LIN {X 0,Y 472.027,Z 1230.388,A -85,B 0,C 180,E1 22778.158,E2 22778.158} C_VEL
LIN {X 0,Y 471.943,Z 1235.002,A -85,B 0,C 180,E1 22775.714,E2 22775.714} C_VEL
LIN {X 0,Y 471.913,Z 1237.961,A -85,B 0,C 180,E1 22773.279,E2 22773.279} C_VEL
LIN {X 0,Y 471.908,Z 1239.363,A -85,B 0,C 180,E1 22770.728,E2 22770.728} C_VEL
LIN {X 0,Y 471.903,Z 1239.099,A -85,B 0,C 180,E1 22768.3,E2 22768.3} C_VEL
LIN {X 0,Y 471.92,Z 1237.256,A -85,B 0,C 180,E1 22765.869,E2 22765.869} C_VEL
LIN {X 0,Y 471.966,Z 1233.719,A -85,B 0,C 180,E1 22763.431,E2 22763.431} C_VEL
LIN {X 0,Y 472.092,Z 1228.265,A -85,B 0,C 180,E1 22760.86,E2 22760.86} C_VEL
LIN {X 0,Y 472.392,Z 1221.418,A -85,B 0,C 180,E1 22758.4,E2 22758.4} C_VEL
LIN {X 0,Y 472.916,Z 1212.648,A -85,B 0,C 180,E1 22755.928,E2 22755.928} C_VEL
LIN {X 0,Y 473.639,Z 1202.902,A -85,B 0,C 180,E1 22753.694,E2 22753.694} C_VEL
LIN {X 0,Y 474.601,Z 1191.85,A -85,B 0,C 180,E1 22751.578,E2 22751.578} C_VEL
LIN {X 0,Y 475.854,Z 1178.616,A -85,B 0,C 180,E1 22749.457,E2 22749.457} C_VEL
LIN {X 0,Y 477.335,Z 1163.705,A -85,B 0,C 180,E1 22747.46,E2 22747.46} C_VEL
LIN {X 0,Y 478.876,Z 1148.153,A -85,B 0,C 180,E1 22745.712,E2 22745.712} C_VEL
LIN {X 0,Y 480.486,Z 1131.656,A -85,B 0,C 180,E1 22744.153,E2 22744.153} C_VEL
LIN {X 0,Y 482.07,Z 1114.027,A -85,B 0,C 180,E1 22742.763,E2 22742.763} C_VEL
LIN {X 0,Y 483.619,Z 1095.064,A -85,B 0,C 180,E1 22741.539,E2 22741.539} C_VEL
LIN {X 0,Y 484.935,Z 1076.494,A -85,B 0,C 180,E1 22740.578,E2 22740.578} C_VEL
LIN {X 0,Y 486.066,Z 1056.533,A -85,B 0,C 180,E1 22739.778,E2 22739.778} C_VEL
LIN {X 0,Y 486.911,Z 1035.363,A -85,B 0,C 180,E1 22739.175,E2 22739.175} C_VEL
LIN {X 0,Y 487.494,Z 1006.649,A -85,B 0,C 180,E1 22738.67,E2 22738.67} C_VEL
LIN {X 0,Y 491.036,Z 793.925,A -85,B 0,C 180,E1 22735.273,E2 22735.273} C_VEL
LIN {X 0,Y 485.904,Z 771.478,A -85,B 0,C 180,E1 22734.421,E2 22734.421} C_VEL
LIN {X 0,Y 487.066,Z 742.84,A -85,B 0,C 180,E1 22731.537,E2 22731.537} C_VEL
LIN {X 0,Y 488.498,Z 716.424,A -85,B 0,C 180,E1 22728.693,E2 22728.693} C_VEL
LIN {X 0,Y 481.564,Z 696.985,A -85,B 0,C 180,E1 22725.751,E2 22725.751} C_VEL
LIN {X 0,Y 475.833,Z 682.945,A -85,B 0,C 180,E1 22723.536,E2 22723.536} C_VEL
LIN {X 0,Y 472.971,Z 675.939,A -85,B 0,C 180,E1 22722.424,E2 22722.424} C_VEL
LIN {X 0,Y 472.97,Z 675.954,A -85,B 0,C 180,E1 22721.46,E2 22721.46} C_VEL
LIN {X 0,Y 474.113,Z 679.098,A -85,B 0,C 180,E1 22720.975,E2 22720.975} C_VEL
LIN {X 0,Y 480.996,Z 694.968,A -85,B 0,C 180,E1 22718.497,E2 22718.497} C_VEL
LIN {X 0,Y 488.174,Z 713.188,A -85,B 0,C 180,E1 22715.858,E2 22715.858} C_VEL
LIN {X 0,Y 489.067,Z 715.897,A -85,B 0,C 180,E1 22715.494,E2 22715.494} C_VEL
LIN {X 0,Y 486.393,Z 754.227,A -85,B 0,C 180,E1 22711.891,E2 22711.891} C_VEL
LIN {X 0,Y 483.773,Z 794.316,A -85,B 0,C 180,E1 22708.182,E2 22708.182} C_VEL
LIN {X 0,Y 481.248,Z 836.985,A -85,B 0,C 180,E1 22704.291,E2 22704.291} C_VEL
LIN {X 0,Y 480.539,Z 852.687,A -85,B 0,C 180,E1 22702.912,E2 22702.912} C_VEL
LIN {X 0,Y 481.743,Z 862.638,A -85,B 0,C 180,E1 22702.654,E2 22702.654} C_VEL
LIN {X 0,Y 478.978,Z 1022.625,A -85,B 0,C 180,E1 22699.905,E2 22699.905} C_VEL
LIN {X 0,Y 478.54,Z 1040.298,A -85,B 0,C 180,E1 22699.368,E2 22699.368} C_VEL
LIN {X 0,Y 477.926,Z 1057.004,A -85,B 0,C 180,E1 22698.634,E2 22698.634} C_VEL
LIN {X 0,Y 477.154,Z 1073.057,A -85,B 0,C 180,E1 22697.689,E2 22697.689} C_VEL
LIN {X 0,Y 476.271,Z 1088.379,A -85,B 0,C 180,E1 22696.527,E2 22696.527} C_VEL
LIN {X 0,Y 475.395,Z 1102.609,A -85,B 0,C 180,E1 22695.18,E2 22695.18} C_VEL
LIN {X 0,Y 474.55,Z 1115.691,A -85,B 0,C 180,E1 22693.65,E2 22693.65} C_VEL
LIN {X 0,Y 473.843,Z 1126.703,A -85,B 0,C 180,E1 22692.058,E2 22692.058} C_VEL
LIN {X 0,Y 473.206,Z 1137.011,A -85,B 0,C 180,E1 22690.224,E2 22690.224} C_VEL
LIN {X 0,Y 472.752,Z 1145.711,A -85,B 0,C 180,E1 22688.269,E2 22688.269} C_VEL
LIN {X 0,Y 472.48,Z 1152.378,A -85,B 0,C 180,E1 22686.318,E2 22686.318} C_VEL
LIN {X 0,Y 472.291,Z 1157.831,A -85,B 0,C 180,E1 22684.128,E2 22684.128} C_VEL
LIN {X 0,Y 472.226,Z 1161.226,A -85,B 0,C 180,E1 22682.011,E2 22682.011} C_VEL
LIN {X 0,Y 472.201,Z 1162.941,A -85,B 0,C 180,E1 22679.879,E2 22679.879} C_VEL
LIN {X 0,Y 472.231,Z 1162.833,A -85,B 0,C 180,E1 22677.573,E2 22677.573} C_VEL
LIN {X 0,Y 472.284,Z 1161.078,A -85,B 0,C 180,E1 22675.508,E2 22675.508} C_VEL
LIN {X 0,Y 472.422,Z 1157.73,A -85,B 0,C 180,E1 22673.438,E2 22673.438} C_VEL
LIN {X 0,Y 472.653,Z 1152.534,A -85,B 0,C 180,E1 22671.362,E2 22671.362} C_VEL
LIN {X 0,Y 473.024,Z 1145.419,A -85,B 0,C 180,E1 22669.28,E2 22669.28} C_VEL
LIN {X 0,Y 473.566,Z 1137.253,A -85,B 0,C 180,E1 22667.44,E2 22667.44} C_VEL
LIN {X 0,Y 474.243,Z 1127.651,A -85,B 0,C 180,E1 22665.72,E2 22665.72} C_VEL
LIN {X 0,Y 474.992,Z 1116.619,A -85,B 0,C 180,E1 22664.119,E2 22664.119} C_VEL
LIN {X 0,Y 475.86,Z 1104.113,A -85,B 0,C 180,E1 22662.641,E2 22662.641} C_VEL
LIN {X 0,Y 476.736,Z 1090.596,A -85,B 0,C 180,E1 22661.347,E2 22661.347} C_VEL
LIN {X 0,Y 477.533,Z 1075.977,A -85,B 0,C 180,E1 22660.236,E2 22660.236} C_VEL
LIN {X 0,Y 478.208,Z 1060.301,A -85,B 0,C 180,E1 22659.308,E2 22659.308} C_VEL
LIN {X 0,Y 478.738,Z 1043.983,A -85,B 0,C 180,E1 22658.586,E2 22658.586} C_VEL
LIN {X 0,Y 479.03,Z 1027.199,A -85,B 0,C 180,E1 22658.081,E2 22658.081} C_VEL
LIN {X 0,Y 481.097,Z 935.545,A -85,B 0,C 180,E1 22656.323,E2 22656.323} C_VEL
LIN {X 0,Y 483.696,Z 869.516,A -85,B 0,C 180,E1 22654.928,E2 22654.928} C_VEL
LIN {X 0,Y 486.372,Z 861.818,A -85,B 0,C 180,E1 22654.359,E2 22654.359} C_VEL
LIN {X 0,Y 491.455,Z 830.458,A -85,B 0,C 180,E1 22650.973,E2 22650.973} C_VEL
LIN {X 0,Y 496.727,Z 807.951,A -85,B 0,C 180,E1 22648.371,E2 22648.371} C_VEL
LIN {X 0,Y 502.512,Z 790.111,A -85,B 0,C 180,E1 22646.143,E2 22646.143} C_VEL
LIN {X 0,Y 508.797,Z 776.41,A -85,B 0,C 180,E1 22644.293,E2 22644.293} C_VEL
LIN {X 0,Y 509.848,Z 774.506,A -85,B 0,C 180,E1 22643.994,E2 22643.994} C_VEL
LIN {X 0,Y 502.789,Z 785.083,A -85,B 0,C 180,E1 22642.698,E2 22642.698} C_VEL
LIN {X 0,Y 498.164,Z 795.448,A -85,B 0,C 180,E1 22641.413,E2 22641.413} C_VEL
LIN {X 0,Y 495.854,Z 805.348,A -85,B 0,C 180,E1 22640.199,E2 22640.199} C_VEL
LIN {X 0,Y 495.553,Z 815.668,A -85,B 0,C 180,E1 22638.956,E2 22638.956} C_VEL
LIN {X 0,Y 497.374,Z 826.582,A -85,B 0,C 180,E1 22637.667,E2 22637.667} C_VEL
LIN {X 0,Y 501.457,Z 837.677,A -85,B 0,C 180,E1 22636.379,E2 22636.379} C_VEL
LIN {X 0,Y 507.651,Z 848.231,A -85,B 0,C 180,E1 22635.158,E2 22635.158} C_VEL
LIN {X 0,Y 515.78,Z 858.073,A -85,B 0,C 180,E1 22634.012,E2 22634.012} C_VEL
LIN {X 0,Y 525.907,Z 867.121,A -85,B 0,C 180,E1 22632.949,E2 22632.949} C_VEL
LIN {X 0,Y 537.102,Z 874.718,A -85,B 0,C 180,E1 22632.032,E2 22632.032} C_VEL
LIN {X 0,Y 549.32,Z 880.935,A -85,B 0,C 180,E1 22631.217,E2 22631.217} C_VEL
LIN {X 0,Y 556.729,Z 883.664,A -85,B 0,C 180,E1 22630.722,E2 22630.722} C_VEL
LIN {X 0,Y 559.457,Z 884.419,A -85,B 0,C 180,E1 22630.458,E2 22630.458} C_VEL
LIN {X 0,Y 556.641,Z 890.597,A -85,B 0,C 180,E1 22630.289,E2 22630.289} C_VEL
LIN {X 0,Y 545.031,Z 908.312,A -85,B 0,C 180,E1 22629.947,E2 22629.947} C_VEL
LIN {X 0,Y 525.372,Z 938.085,A -85,B 0,C 180,E1 22629.116,E2 22629.116} C_VEL
LIN {X 0,Y 515.376,Z 955.996,A -85,B 0,C 180,E1 22628.518,E2 22628.518} C_VEL
LIN {X 0,Y 509.372,Z 970.036,A -85,B 0,C 180,E1 22627.98,E2 22627.98} C_VEL
LIN {X 0,Y 506.831,Z 975.536,A -85,B 0,C 180,E1 22627.774,E2 22627.774} C_VEL
LIN {X 0,Y 500.091,Z 990.21,A -85,B 0,C 180,E1 22627.215,E2 22627.215} C_VEL
LIN {X 0,Y 492.099,Z 1013.905,A -85,B 0,C 180,E1 22626.175,E2 22626.175} C_VEL
LIN {X 0,Y 490.679,Z 1019.518,A -85,B 0,C 180,E1 22625.946,E2 22625.946} C_VEL
LIN {X 0,Y 490.022,Z 1029.861,A -85,B 0,C 180,E1 22625.815,E2 22625.815} C_VEL
LIN {X 0,Y 489.453,Z 1064.268,A -85,B 0,C 180,E1 22625.251,E2 22625.251} C_VEL
LIN {X 0,Y 488.525,Z 1088.169,A -85,B 0,C 180,E1 22624.651,E2 22624.651} C_VEL
LIN {X 0,Y 487.384,Z 1111.453,A -85,B 0,C 180,E1 22623.84,E2 22623.84} C_VEL
LIN {X 0,Y 486.067,Z 1134.154,A -85,B 0,C 180,E1 22622.822,E2 22622.822} C_VEL
LIN {X 0,Y 484.559,Z 1155.984,A -85,B 0,C 180,E1 22621.609,E2 22621.609} C_VEL
LIN {X 0,Y 482.968,Z 1176.918,A -85,B 0,C 180,E1 22620.204,E2 22620.204} C_VEL
LIN {X 0,Y 481.619,Z 1192.738,A -85,B 0,C 180,E1 22618.929,E2 22618.929} C_VEL
LIN {X 0,Y 480.163,Z 1206.829,A -85,B 0,C 180,E1 22617.535,E2 22617.535} C_VEL
LIN {X 0,Y 478.573,Z 1221.087,A -85,B 0,C 180,E1 22615.891,E2 22615.891} C_VEL
LIN {X 0,Y 477.202,Z 1233.662,A -85,B 0,C 180,E1 22614.247,E2 22614.247} C_VEL
LIN {X 0,Y 475.743,Z 1248.075,A -85,B 0,C 180,E1 22612.099,E2 22612.099} C_VEL
LIN {X 0,Y 474.509,Z 1260.921,A -85,B 0,C 180,E1 22609.832,E2 22609.832} C_VEL
LIN {X 0,Y 473.67,Z 1270.78,A -85,B 0,C 180,E1 22607.823,E2 22607.823} C_VEL
LIN {X 0,Y 472.974,Z 1280.325,A -85,B 0,C 180,E1 22605.574,E2 22605.574} C_VEL
LIN {X 0,Y 472.429,Z 1289.877,A -85,B 0,C 180,E1 22602.84,E2 22602.84} C_VEL
LIN {X 0,Y 472.149,Z 1296.436,A -85,B 0,C 180,E1 22600.494,E2 22600.494} C_VEL
LIN {X 0,Y 471.998,Z 1301.632,A -85,B 0,C 180,E1 22598.16,E2 22598.16} C_VEL
LIN {X 0,Y 471.927,Z 1306.121,A -85,B 0,C 180,E1 22595.349,E2 22595.349} C_VEL
LIN {X 0,Y 471.903,Z 1308.434,A -85,B 0,C 180,E1 22592.915,E2 22592.915} C_VEL
LIN {X 0,Y 471.896,Z 1309.388,A -85,B 0,C 180,E1 22590.608,E2 22590.608} C_VEL
LIN {X 0,Y 471.908,Z 1308.917,A -85,B 0,C 180,E1 22587.815,E2 22587.815} C_VEL
LIN {X 0,Y 471.918,Z 1306.943,A -85,B 0,C 180,E1 22585.383,E2 22585.383} C_VEL
LIN {X 0,Y 471.961,Z 1303.794,A -85,B 0,C 180,E1 22583.065,E2 22583.065} C_VEL
LIN {X 0,Y 472.071,Z 1299.112,A -85,B 0,C 180,E1 22580.614,E2 22580.614} C_VEL
LIN {X 0,Y 472.324,Z 1292.113,A -85,B 0,C 180,E1 22577.903,E2 22577.903} C_VEL
LIN {X 0,Y 472.718,Z 1284.471,A -85,B 0,C 180,E1 22575.548,E2 22575.548} C_VEL
LIN {X 0,Y 473.375,Z 1274.765,A -85,B 0,C 180,E1 22573.054,E2 22573.054} C_VEL
LIN {X 0,Y 474.273,Z 1263.528,A -85,B 0,C 180,E1 22570.672,E2 22570.672} C_VEL
LIN {X 0,Y 475.286,Z 1252.524,A -85,B 0,C 180,E1 22568.658,E2 22568.658} C_VEL
LIN {X 0,Y 476.669,Z 1239.071,A -85,B 0,C 180,E1 22566.514,E2 22566.514} C_VEL
LIN {X 0,Y 478.346,Z 1223.146,A -85,B 0,C 180,E1 22564.363,E2 22564.363} C_VEL
LIN {X 0,Y 479.836,Z 1209.702,A -85,B 0,C 180,E1 22562.782,E2 22562.782} C_VEL
LIN {X 0,Y 481.31,Z 1196.28,A -85,B 0,C 180,E1 22561.392,E2 22561.392} C_VEL
LIN {X 0,Y 483.032,Z 1177.605,A -85,B 0,C 180,E1 22559.802,E2 22559.802} C_VEL
LIN {X 0,Y 484.805,Z 1157.277,A -85,B 0,C 180,E1 22558.341,E2 22558.341} C_VEL
LIN {X 0,Y 486.575,Z 1135.76,A -85,B 0,C 180,E1 22557.055,E2 22557.055} C_VEL
LIN {X 0,Y 488.148,Z 1114.091,A -85,B 0,C 180,E1 22556.002,E2 22556.002} C_VEL
LIN {X 0,Y 489.575,Z 1091.135,A -85,B 0,C 180,E1 22555.128,E2 22555.128} C_VEL
LIN {X 0,Y 490.74,Z 1068.207,A -85,B 0,C 180,E1 22554.494,E2 22554.494} C_VEL
LIN {X 0,Y 491.441,Z 1041.848,A -85,B 0,C 180,E1 22554.015,E2 22554.015} C_VEL
LIN {X 0,Y 492.099,Z 1021.688,A -85,B 0,C 180,E1 22553.682,E2 22553.682} C_VEL
LIN {X 0,Y 497.028,Z 1006.052,A -85,B 0,C 180,E1 22552.952,E2 22552.952} C_VEL
LIN {X 0,Y 503.429,Z 988.405,A -85,B 0,C 180,E1 22552.208,E2 22552.208} C_VEL
LIN {X 0,Y 510.583,Z 973.055,A -85,B 0,C 180,E1 22551.7,E2 22551.7} C_VEL
LIN {X 0,Y 516.137,Z 959.333,A -85,B 0,C 180,E1 22551.195,E2 22551.195} C_VEL
LIN {X 0,Y 524.952,Z 942.125,A -85,B 0,C 180,E1 22550.707,E2 22550.707} C_VEL
LIN {X 0,Y 541.254,Z 914.948,A -85,B 0,C 180,E1 22550.133,E2 22550.133} C_VEL
LIN {X 0,Y 557.706,Z 888.615,A -85,B 0,C 180,E1 22549.67,E2 22549.67} C_VEL
LIN {X 0,Y 559.402,Z 884.287,A -85,B 0,C 180,E1 22549.528,E2 22549.528} C_VEL
LIN {X 0,Y 547.093,Z 880.541,A -85,B 0,C 180,E1 22548.372,E2 22548.372} C_VEL
LIN {X 0,Y 536.038,Z 875.106,A -85,B 0,C 180,E1 22547.143,E2 22547.143} C_VEL
LIN {X 0,Y 526.595,Z 868.26,A -85,B 0,C 180,E1 22545.866,E2 22545.866} C_VEL
LIN {X 0,Y 518.671,Z 860.097,A -85,B 0,C 180,E1 22544.563,E2 22544.563} C_VEL
LIN {X 0,Y 512.248,Z 850.667,A -85,B 0,C 180,E1 22543.245,E2 22543.245} C_VEL
LIN {X 0,Y 507.136,Z 839.468,A -85,B 0,C 180,E1 22541.865,E2 22541.865} C_VEL
LIN {X 0,Y 503.479,Z 826.201,A -85,B 0,C 180,E1 22540.42,E2 22540.42} C_VEL
LIN {X 0,Y 501.504,Z 811.016,A -85,B 0,C 180,E1 22538.964,E2 22538.964} C_VEL
LIN {X 0,Y 501.31,Z 794.305,A -85,B 0,C 180,E1 22537.54,E2 22537.54} C_VEL
LIN {X 0,Y 505.763,Z 740.56,A -85,B 0,C 180,E1 22533.413,E2 22533.413} C_VEL
LIN {X 0,Y 506.021,Z 736.154,A -85,B 0,C 180,E1 22533.049,E2 22533.049} C_VEL
LIN {X 0,Y 496.27,Z 718.046,A -85,B 0,C 180,E1 22529.977,E2 22529.977} C_VEL
LIN {X 0,Y 488.915,Z 704.66,A -85,B 0,C 180,E1 22527.528,E2 22527.528} C_VEL
LIN {X 0,Y 483.047,Z 694.382,A -85,B 0,C 180,E1 22525.501,E2 22525.501} C_VEL
LIN {X 0,Y 480.533,Z 689.941,A -85,B 0,C 180,E1 22524.591,E2 22524.591} C_VEL
LIN {X 0,Y 478.059,Z 685.483,A -85,B 0,C 180,E1 22523.676,E2 22523.676} C_VEL
LIN {X 0,Y 475.958,Z 681.627,A -85,B 0,C 180,E1 22522.869,E2 22522.869} C_VEL
LIN {X 0,Y 473.409,Z 677.657,A -85,B 0,C 180,E1 22521.952,E2 22521.952} C_VEL
LIN {X 0,Y 472.947,Z 675.821,A -85,B 0,C 180,E1 22521.648,E2 22521.648} C_VEL
LIN {X 0,Y 472.954,Z 675.824,A -85,B 0,C 180,E1 22517.978,E2 22517.978} C_VEL
LIN {X 0,Y 472.946,Z 675.824,A -85,B 0,C 180,E1 22514.321,E2 22514.321} C_VEL
LIN {X 0,Y 472.947,Z 675.824,A -85,B 0,C 180,E1 22510.722,E2 22510.722} C_VEL
LIN {X 0,Y 472.958,Z 675.82,A -85,B 0,C 180,E1 22507.043,E2 22507.043} C_VEL
LIN {X 0,Y 472.941,Z 675.824,A -85,B 0,C 180,E1 22503.393,E2 22503.393} C_VEL
LIN {X 0,Y 472.954,Z 675.821,A -85,B 0,C 180,E1 22499.757,E2 22499.757} C_VEL
LIN {X 0,Y 472.947,Z 675.821,A -85,B 0,C 180,E1 22496.121,E2 22496.121} C_VEL
LIN {X 0,Y 472.937,Z 675.825,A -85,B 0,C 180,E1 22492.468,E2 22492.468} C_VEL
LIN {X 0,Y 472.95,Z 675.822,A -85,B 0,C 180,E1 22488.908,E2 22488.908} C_VEL
LIN {X 0,Y 472.949,Z 675.823,A -85,B 0,C 180,E1 22485.304,E2 22485.304} C_VEL
LIN {X 0,Y 472.939,Z 675.821,A -85,B 0,C 180,E1 22481.639,E2 22481.639} C_VEL
LIN {X 0,Y 472.957,Z 675.821,A -85,B 0,C 180,E1 22478.026,E2 22478.026} C_VEL
LIN {X 0,Y 472.942,Z 675.823,A -85,B 0,C 180,E1 22474.316,E2 22474.316} C_VEL
LIN {X 0,Y 472.936,Z 675.784,A -85,B 0,C 180,E1 22470.766,E2 22470.766} C_VEL
LIN {X 0,Y 472.954,Z 675.822,A -85,B 0,C 180,E1 22467.234,E2 22467.234} C_VEL
LIN {X 0,Y 472.938,Z 675.8,A -85,B 0,C 180,E1 22463.553,E2 22463.553} C_VEL
LIN {X 0,Y 472.938,Z 675.802,A -85,B 0,C 180,E1 22460.006,E2 22460.006} C_VEL
LIN {X 0,Y 472.951,Z 675.825,A -85,B 0,C 180,E1 22456.433,E2 22456.433} C_VEL
LIN {X 0,Y 472.966,Z 675.939,A -85,B 0,C 180,E1 22454.184,E2 22454.184} C_VEL
LIN {X 0,Y 474.014,Z 678.945,A -85,B 0,C 180,E1 22453.83,E2 22453.83} C_VEL
LIN {X 0,Y 475.481,Z 681.845,A -85,B 0,C 180,E1 22453.442,E2 22453.442} C_VEL
LIN {X 0,Y 483.15,Z 698.3,A -85,B 0,C 180,E1 22451.304,E2 22451.304} C_VEL
LIN {X 0,Y 490.743,Z 716.812,A -85,B 0,C 180,E1 22449.08,E2 22449.08} C_VEL
LIN {X 0,Y 488.698,Z 760.843,A -85,B 0,C 180,E1 22445.884,E2 22445.884} C_VEL
LIN {X 0,Y 488.556,Z 770.502,A -85,B 0,C 180,E1 22445.256,E2 22445.256} C_VEL
LIN {X 0,Y 489.009,Z 773.268,A -85,B 0,C 180,E1 22445.169,E2 22445.169} C_VEL
LIN {X 0,Y 489.235,Z 779.807,A -85,B 0,C 180,E1 22445.034,E2 22445.034} C_VEL
LIN {X 0,Y 487.638,Z 789.743,A -85,B 0,C 180,E1 22444.991,E2 22444.991} C_VEL
LIN {X 0,Y 484.595,Z 804.217,A -85,B 0,C 180,E1 22444.989,E2 22444.989} C_VEL
LIN {X 0,Y 484.245,Z 808.717,A -85,B 0,C 180,E1 22444.938,E2 22444.938} C_VEL
LIN {X 0,Y 480.185,Z 1031.487,A -85,B 0,C 180,E1 22441.312,E2 22441.312} C_VEL
LIN {X 0,Y 479.366,Z 1052.367,A -85,B 0,C 180,E1 22440.762,E2 22440.762} C_VEL
LIN {X 0,Y 478.234,Z 1073.043,A -85,B 0,C 180,E1 22439.978,E2 22439.978} C_VEL
LIN {X 0,Y 476.872,Z 1092.041,A -85,B 0,C 180,E1 22439.034,E2 22439.034} C_VEL
LIN {X 0,Y 475.373,Z 1110.231,A -85,B 0,C 180,E1 22437.903,E2 22437.903} C_VEL
LIN {X 0,Y 473.655,Z 1128.403,A -85,B 0,C 180,E1 22436.516,E2 22436.516} C_VEL
LIN {X 0,Y 471.885,Z 1145.616,A -85,B 0,C 180,E1 22434.923,E2 22434.923} C_VEL
LIN {X 0,Y 470.228,Z 1160.946,A -85,B 0,C 180,E1 22433.23,E2 22433.23} C_VEL
LIN {X 0,Y 468.703,Z 1175.051,A -85,B 0,C 180,E1 22431.394,E2 22431.394} C_VEL
LIN {X 0,Y 467.317,Z 1188.383,A -85,B 0,C 180,E1 22429.342,E2 22429.342} C_VEL
LIN {X 0,Y 466.197,Z 1200.038,A -85,B 0,C 180,E1 22427.215,E2 22427.215} C_VEL
LIN {X 0,Y 465.312,Z 1210.434,A -85,B 0,C 180,E1 22424.942,E2 22424.942} C_VEL
LIN {X 0,Y 464.634,Z 1219.787,A -85,B 0,C 180,E1 22422.426,E2 22422.426} C_VEL
LIN {X 0,Y 464.237,Z 1227.132,A -85,B 0,C 180,E1 22419.921,E2 22419.921} C_VEL
LIN {X 0,Y 464.022,Z 1232.679,A -85,B 0,C 180,E1 22417.428,E2 22417.428} C_VEL
LIN {X 0,Y 463.939,Z 1236.571,A -85,B 0,C 180,E1 22414.945,E2 22414.945} C_VEL
LIN {X 0,Y 463.918,Z 1238.909,A -85,B 0,C 180,E1 22412.47,E2 22412.47} C_VEL
LIN {X 0,Y 463.917,Z 1239.729,A -85,B 0,C 180,E1 22409.999,E2 22409.999} C_VEL
LIN {X 0,Y 463.915,Z 1238.892,A -85,B 0,C 180,E1 22407.405,E2 22407.405} C_VEL
LIN {X 0,Y 463.94,Z 1236.53,A -85,B 0,C 180,E1 22404.93,E2 22404.93} C_VEL
LIN {X 0,Y 464.039,Z 1232.365,A -85,B 0,C 180,E1 22402.322,E2 22402.322} C_VEL
LIN {X 0,Y 464.255,Z 1226.654,A -85,B 0,C 180,E1 22399.814,E2 22399.814} C_VEL
LIN {X 0,Y 464.645,Z 1219.655,A -85,B 0,C 180,E1 22397.447,E2 22397.447} C_VEL
LIN {X 0,Y 465.28,Z 1210.794,A -85,B 0,C 180,E1 22395.056,E2 22395.056} C_VEL
LIN {X 0,Y 466.216,Z 1199.849,A -85,B 0,C 180,E1 22392.656,E2 22392.656} C_VEL
LIN {X 0,Y 467.356,Z 1188.005,A -85,B 0,C 180,E1 22390.503,E2 22390.503} C_VEL
LIN {X 0,Y 468.736,Z 1174.764,A -85,B 0,C 180,E1 22388.475,E2 22388.475} C_VEL
LIN {X 0,Y 470.373,Z 1159.524,A -85,B 0,C 180,E1 22386.511,E2 22386.511} C_VEL
LIN {X 0,Y 472.158,Z 1142.897,A -85,B 0,C 180,E1 22384.72,E2 22384.72} C_VEL
LIN {X 0,Y 473.89,Z 1125.851,A -85,B 0,C 180,E1 22383.188,E2 22383.188} C_VEL
LIN {X 0,Y 475.513,Z 1108.664,A -85,B 0,C 180,E1 22381.9,E2 22381.9} C_VEL
LIN {X 0,Y 477.041,Z 1090.144,A -85,B 0,C 180,E1 22380.767,E2 22380.767} C_VEL
LIN {X 0,Y 478.393,Z 1070.604,A -85,B 0,C 180,E1 22379.824,E2 22379.824} C_VEL
LIN {X 0,Y 479.447,Z 1050.707,A -85,B 0,C 180,E1 22379.095,E2 22379.095} C_VEL
LIN {X 0,Y 480.227,Z 1029.772,A -85,B 0,C 180,E1 22378.563,E2 22378.563} C_VEL
LIN {X 0,Y 484.468,Z 796.881,A -85,B 0,C 180,E1 22374.778,E2 22374.778} C_VEL
LIN {X 0,Y 483.819,Z 792.472,A -85,B 0,C 180,E1 22374.644,E2 22374.644} C_VEL
LIN {X 0,Y 479.103,Z 772.305,A -85,B 0,C 180,E1 22373.867,E2 22373.867} C_VEL
LIN {X 0,Y 480.243,Z 745.321,A -85,B 0,C 180,E1 22371.139,E2 22371.139} C_VEL
LIN {X 0,Y 481.659,Z 719.994,A -85,B 0,C 180,E1 22368.408,E2 22368.408} C_VEL
LIN {X 0,Y 474.936,Z 701.008,A -85,B 0,C 180,E1 22365.488,E2 22365.488} C_VEL
LIN {X 0,Y 469.094,Z 686.695,A -85,B 0,C 180,E1 22363.173,E2 22363.173} C_VEL
LIN {X 0,Y 466.014,Z 679.803,A -85,B 0,C 180,E1 22362.022,E2 22362.022} C_VEL
LIN {X 0,Y 465.799,Z 679.402,A -85,B 0,C 180,E1 22361.922,E2 22361.922} C_VEL
LIN {X 0,Y 468.625,Z 685.422,A -85,B 0,C 180,E1 22360.921,E2 22360.921} C_VEL
LIN {X 0,Y 476.2,Z 703.373,A -85,B 0,C 180,E1 22358.12,E2 22358.12} C_VEL
LIN {X 0,Y 482.247,Z 719.132,A -85,B 0,C 180,E1 22355.838,E2 22355.838} C_VEL
LIN {X 0,Y 479.481,Z 756.766,A -85,B 0,C 180,E1 22352.265,E2 22352.265} C_VEL
LIN {X 0,Y 476.721,Z 797.118,A -85,B 0,C 180,E1 22348.502,E2 22348.502} C_VEL
LIN {X 0,Y 474.03,Z 840.018,A -85,B 0,C 180,E1 22344.553,E2 22344.553} C_VEL
LIN {X 0,Y 473.384,Z 853.662,A -85,B 0,C 180,E1 22343.346,E2 22343.346} C_VEL
LIN {X 0,Y 474.617,Z 863.66,A -85,B 0,C 180,E1 22343.08,E2 22343.08} C_VEL
LIN {X 0,Y 471.533,Z 1023.957,A -85,B 0,C 180,E1 22340.237,E2 22340.237} C_VEL
LIN {X 0,Y 471.066,Z 1041.841,A -85,B 0,C 180,E1 22339.678,E2 22339.678} C_VEL
LIN {X 0,Y 470.411,Z 1058.633,A -85,B 0,C 180,E1 22338.92,E2 22338.92} C_VEL
LIN {X 0,Y 469.617,Z 1074.222,A -85,B 0,C 180,E1 22337.982,E2 22337.982} C_VEL
LIN {X 0,Y 468.688,Z 1089.54,A -85,B 0,C 180,E1 22336.802,E2 22336.802} C_VEL
LIN {X 0,Y 467.742,Z 1104.057,A -85,B 0,C 180,E1 22335.405,E2 22335.405} C_VEL
LIN {X 0,Y 466.863,Z 1116.877,A -85,B 0,C 180,E1 22333.879,E2 22333.879} C_VEL
LIN {X 0,Y 466.052,Z 1128.661,A -85,B 0,C 180,E1 22332.137,E2 22332.137} C_VEL
LIN {X 0,Y 465.379,Z 1138.912,A -85,B 0,C 180,E1 22330.26,E2 22330.26} C_VEL
LIN {X 0,Y 464.906,Z 1147.444,A -85,B 0,C 180,E1 22328.285,E2 22328.285} C_VEL
LIN {X 0,Y 464.61,Z 1154.011,A -85,B 0,C 180,E1 22326.301,E2 22326.301} C_VEL
LIN {X 0,Y 464.413,Z 1159.383,A -85,B 0,C 180,E1 22324.074,E2 22324.074} C_VEL
LIN {X 0,Y 464.347,Z 1162.671,A -85,B 0,C 180,E1 22321.975,E2 22321.975} C_VEL
LIN {X 0,Y 464.315,Z 1164.341,A -85,B 0,C 180,E1 22319.754,E2 22319.754} C_VEL
LIN {X 0,Y 464.357,Z 1164.225,A -85,B 0,C 180,E1 22317.532,E2 22317.532} C_VEL
LIN {X 0,Y 464.434,Z 1162.369,A -85,B 0,C 180,E1 22315.308,E2 22315.308} C_VEL
LIN {X 0,Y 464.606,Z 1158.885,A -85,B 0,C 180,E1 22313.203,E2 22313.203} C_VEL
LIN {X 0,Y 464.875,Z 1153.599,A -85,B 0,C 180,E1 22311.092,E2 22311.092} C_VEL
LIN {X 0,Y 465.277,Z 1146.852,A -85,B 0,C 180,E1 22309.1,E2 22309.1} C_VEL
LIN {X 0,Y 465.875,Z 1138.685,A -85,B 0,C 180,E1 22307.229,E2 22307.229} C_VEL
LIN {X 0,Y 466.605,Z 1129.054,A -85,B 0,C 180,E1 22305.481,E2 22305.481} C_VEL
LIN {X 0,Y 467.434,Z 1117.833,A -85,B 0,C 180,E1 22303.829,E2 22303.829} C_VEL
LIN {X 0,Y 468.348,Z 1105.516,A -85,B 0,C 180,E1 22302.353,E2 22302.353} C_VEL
LIN {X 0,Y 469.271,Z 1091.941,A -85,B 0,C 180,E1 22301.039,E2 22301.039} C_VEL
LIN {X 0,Y 470.105,Z 1077.235,A -85,B 0,C 180,E1 22299.911,E2 22299.911} C_VEL
LIN {X 0,Y 470.816,Z 1061.527,A -85,B 0,C 180,E1 22298.968,E2 22298.968} C_VEL
LIN {X 0,Y 471.364,Z 1045.098,A -85,B 0,C 180,E1 22298.235,E2 22298.235} C_VEL
LIN {X 0,Y 471.631,Z 1028.071,A -85,B 0,C 180,E1 22297.728,E2 22297.728} C_VEL
LIN {X 0,Y 473.725,Z 946.531,A -85,B 0,C 180,E1 22296.082,E2 22296.082} C_VEL
LIN {X 0,Y 477.011,Z 873.239,A -85,B 0,C 180,E1 22294.452,E2 22294.452} C_VEL
LIN {X 0,Y 480.344,Z 864.427,A -85,B 0,C 180,E1 22293.814,E2 22293.814} C_VEL
LIN {X 0,Y 485.823,Z 834.197,A -85,B 0,C 180,E1 22290.468,E2 22290.468} C_VEL
LIN {X 0,Y 491.406,Z 812.773,A -85,B 0,C 180,E1 22287.924,E2 22287.924} C_VEL
LIN {X 0,Y 497.492,Z 795.879,A -85,B 0,C 180,E1 22285.755,E2 22285.755} C_VEL
LIN {X 0,Y 503.476,Z 783.89,A -85,B 0,C 180,E1 22284.077,E2 22284.077} C_VEL
LIN {X 0,Y 496.703,Z 794.089,A -85,B 0,C 180,E1 22282.763,E2 22282.763} C_VEL
LIN {X 0,Y 492.237,Z 804.337,A -85,B 0,C 180,E1 22281.421,E2 22281.421} C_VEL
LIN {X 0,Y 490.22,Z 813.866,A -85,B 0,C 180,E1 22280.176,E2 22280.176} C_VEL
LIN {X 0,Y 490.215,Z 824.17,A -85,B 0,C 180,E1 22278.862,E2 22278.862} C_VEL
LIN {X 0,Y 492.409,Z 834.813,A -85,B 0,C 180,E1 22277.534,E2 22277.534} C_VEL
LIN {X 0,Y 496.547,Z 844.948,A -85,B 0,C 180,E1 22276.294,E2 22276.294} C_VEL
LIN {X 0,Y 502.848,Z 855.102,A -85,B 0,C 180,E1 22275.062,E2 22275.062} C_VEL
LIN {X 0,Y 511.555,Z 865.187,A -85,B 0,C 180,E1 22273.844,E2 22273.844} C_VEL
LIN {X 0,Y 521.716,Z 873.932,A -85,B 0,C 180,E1 22272.777,E2 22272.777} C_VEL
LIN {X 0,Y 532.924,Z 881.364,A -85,B 0,C 180,E1 22271.855,E2 22271.855} C_VEL
LIN {X 0,Y 545.803,Z 887.827,A -85,B 0,C 180,E1 22270.997,E2 22270.997} C_VEL
LIN {X 0,Y 549.692,Z 889.544,A -85,B 0,C 180,E1 22270.749,E2 22270.749} C_VEL
LIN {X 0,Y 522.34,Z 929.728,A -85,B 0,C 180,E1 22269.691,E2 22269.691} C_VEL
LIN {X 0,Y 511.26,Z 948.594,A -85,B 0,C 180,E1 22269.103,E2 22269.103} C_VEL
LIN {X 0,Y 503.934,Z 964.141,A -85,B 0,C 180,E1 22268.537,E2 22268.537} C_VEL
LIN {X 0,Y 500.848,Z 971.749,A -85,B 0,C 180,E1 22268.234,E2 22268.234} C_VEL
LIN {X 0,Y 493.91,Z 986.276,A -85,B 0,C 180,E1 22267.688,E2 22267.688} C_VEL
LIN {X 0,Y 484.729,Z 1012.865,A -85,B 0,C 180,E1 22266.52,E2 22266.52} C_VEL
LIN {X 0,Y 483.666,Z 1017.158,A -85,B 0,C 180,E1 22266.351,E2 22266.351} C_VEL
LIN {X 0,Y 482.711,Z 1028.266,A -85,B 0,C 180,E1 22266.22,E2 22266.22} C_VEL
LIN {X 0,Y 482.065,Z 1063.174,A -85,B 0,C 180,E1 22265.629,E2 22265.629} C_VEL
LIN {X 0,Y 481.074,Z 1087.093,A -85,B 0,C 180,E1 22265.013,E2 22265.013} C_VEL
LIN {X 0,Y 479.836,Z 1110.406,A -85,B 0,C 180,E1 22264.183,E2 22264.183} C_VEL
LIN {X 0,Y 478.437,Z 1133.531,A -85,B 0,C 180,E1 22263.127,E2 22263.127} C_VEL
LIN {X 0,Y 476.799,Z 1156.143,A -85,B 0,C 180,E1 22261.843,E2 22261.843} C_VEL
LIN {X 0,Y 475.072,Z 1177.888,A -85,B 0,C 180,E1 22260.339,E2 22260.339} C_VEL
LIN {X 0,Y 473.361,Z 1197.738,A -85,B 0,C 180,E1 22258.692,E2 22258.692} C_VEL
LIN {X 0,Y 471.604,Z 1216.476,A -85,B 0,C 180,E1 22256.846,E2 22256.846} C_VEL
LIN {X 0,Y 470.137,Z 1229.993,A -85,B 0,C 180,E1 22255.173,E2 22255.173} C_VEL
LIN {X 0,Y 468.617,Z 1243.162,A -85,B 0,C 180,E1 22253.249,E2 22253.249} C_VEL
LIN {X 0,Y 467.382,Z 1254.703,A -85,B 0,C 180,E1 22251.327,E2 22251.327} C_VEL
LIN {X 0,Y 466.175,Z 1267.336,A -85,B 0,C 180,E1 22248.897,E2 22248.897} C_VEL
LIN {X 0,Y 465.274,Z 1277.811,A -85,B 0,C 180,E1 22246.479,E2 22246.479} C_VEL
LIN {X 0,Y 464.696,Z 1286.206,A -85,B 0,C 180,E1 22244.199,E2 22244.199} C_VEL
LIN {X 0,Y 464.272,Z 1294.373,A -85,B 0,C 180,E1 22241.511,E2 22241.511} C_VEL
LIN {X 0,Y 464.044,Z 1300.379,A -85,B 0,C 180,E1 22238.925,E2 22238.925} C_VEL
LIN {X 0,Y 463.957,Z 1304.373,A -85,B 0,C 180,E1 22236.683,E2 22236.683} C_VEL
LIN {X 0,Y 463.906,Z 1307.611,A -85,B 0,C 180,E1 22234.079,E2 22234.079} C_VEL
LIN {X 0,Y 463.903,Z 1309.223,A -85,B 0,C 180,E1 22231.359,E2 22231.359} C_VEL
LIN {X 0,Y 463.902,Z 1309.33,A -85,B 0,C 180,E1 22229.136,E2 22229.136} C_VEL
LIN {X 0,Y 463.91,Z 1308.264,A -85,B 0,C 180,E1 22226.788,E2 22226.788} C_VEL
LIN {X 0,Y 463.933,Z 1305.67,A -85,B 0,C 180,E1 22224.187,E2 22224.187} C_VEL
LIN {X 0,Y 464.012,Z 1301.263,A -85,B 0,C 180,E1 22221.514,E2 22221.514} C_VEL
LIN {X 0,Y 464.171,Z 1296.439,A -85,B 0,C 180,E1 22219.325,E2 22219.325} C_VEL
LIN {X 0,Y 464.461,Z 1290.24,A -85,B 0,C 180,E1 22217.063,E2 22217.063} C_VEL
LIN {X 0,Y 465.023,Z 1281.343,A -85,B 0,C 180,E1 22214.41,E2 22214.41} C_VEL
LIN {X 0,Y 465.806,Z 1271.247,A -85,B 0,C 180,E1 22211.971,E2 22211.971} C_VEL
LIN {X 0,Y 466.699,Z 1261.57,A -85,B 0,C 180,E1 22209.954,E2 22209.954} C_VEL
LIN {X 0,Y 468.021,Z 1248.853,A -85,B 0,C 180,E1 22207.65,E2 22207.65} C_VEL
LIN {X 0,Y 469.584,Z 1234.585,A -85,B 0,C 180,E1 22205.469,E2 22205.469} C_VEL
LIN {X 0,Y 470.908,Z 1223.026,A -85,B 0,C 180,E1 22203.928,E2 22203.928} C_VEL
LIN {X 0,Y 472.258,Z 1209.86,A -85,B 0,C 180,E1 22202.445,E2 22202.445} C_VEL
LIN {X 0,Y 473.986,Z 1192.924,A -85,B 0,C 180,E1 22200.769,E2 22200.769} C_VEL
LIN {X 0,Y 475.964,Z 1172.943,A -85,B 0,C 180,E1 22199.094,E2 22199.094} C_VEL
LIN {X 0,Y 477.925,Z 1151.492,A -85,B 0,C 180,E1 22197.578,E2 22197.578} C_VEL
LIN {X 0,Y 479.785,Z 1130.104,A -85,B 0,C 180,E1 22196.336,E2 22196.336} C_VEL
LIN {X 0,Y 481.424,Z 1108.409,A -85,B 0,C 180,E1 22195.316,E2 22195.316} C_VEL
LIN {X 0,Y 482.905,Z 1085.731,A -85,B 0,C 180,E1 22194.496,E2 22194.496} C_VEL
LIN {X 0,Y 484.082,Z 1062.431,A -85,B 0,C 180,E1 22193.885,E2 22193.885} C_VEL
LIN {X 0,Y 485.332,Z 1021.058,A -85,B 0,C 180,E1 22193.185,E2 22193.185} C_VEL
LIN {X 0,Y 490.413,Z 1005.176,A -85,B 0,C 180,E1 22192.44,E2 22192.44} C_VEL
LIN {X 0,Y 497.119,Z 987.073,A -85,B 0,C 180,E1 22191.666,E2 22191.666} C_VEL
LIN {X 0,Y 504.393,Z 971.412,A -85,B 0,C 180,E1 22191.143,E2 22191.143} C_VEL
LIN {X 0,Y 510.505,Z 956.741,A -85,B 0,C 180,E1 22190.612,E2 22190.612} C_VEL
LIN {X 0,Y 519.912,Z 938.695,A -85,B 0,C 180,E1 22190.114,E2 22190.114} C_VEL
LIN {X 0,Y 537.621,Z 909.465,A -85,B 0,C 180,E1 22189.521,E2 22189.521} C_VEL
LIN {X 0,Y 550.018,Z 889.734,A -85,B 0,C 180,E1 22189.173,E2 22189.173} C_VEL
LIN {X 0,Y 538.211,Z 885.219,A -85,B 0,C 180,E1 22187.996,E2 22187.996} C_VEL
LIN {X 0,Y 527.508,Z 879.073,A -85,B 0,C 180,E1 22186.706,E2 22186.706} C_VEL
LIN {X 0,Y 517.814,Z 871.02,A -85,B 0,C 180,E1 22185.282,E2 22185.282} C_VEL
LIN {X 0,Y 509.805,Z 861.361,A -85,B 0,C 180,E1 22183.814,E2 22183.814} C_VEL
LIN {X 0,Y 503.895,Z 850.978,A -85,B 0,C 180,E1 22182.426,E2 22182.426} C_VEL
LIN {X 0,Y 499.374,Z 838.84,A -85,B 0,C 180,E1 22180.99,E2 22180.99} C_VEL
LIN {X 0,Y 496.349,Z 824.685,A -85,B 0,C 180,E1 22179.51,E2 22179.51} C_VEL
LIN {X 0,Y 495.056,Z 808.748,A -85,B 0,C 180,E1 22178.025,E2 22178.025} C_VEL
LIN {X 0,Y 495.629,Z 788.954,A -85,B 0,C 180,E1 22176.398,E2 22176.398} C_VEL
LIN {X 0,Y 499.643,Z 746.305,A -85,B 0,C 180,E1 22173.114,E2 22173.114} C_VEL
LIN {X 0,Y 500.116,Z 740.794,A -85,B 0,C 180,E1 22172.67,E2 22172.67} C_VEL
LIN {X 0,Y 491.078,Z 723.911,A -85,B 0,C 180,E1 22169.788,E2 22169.788} C_VEL
LIN {X 0,Y 483.404,Z 709.96,A -85,B 0,C 180,E1 22167.2,E2 22167.2} C_VEL
LIN {X 0,Y 476.068,Z 696.707,A -85,B 0,C 180,E1 22164.572,E2 22164.572} C_VEL
LIN {X 0,Y 472.541,Z 690.858,A -85,B 0,C 180,E1 22163.308,E2 22163.308} C_VEL
LIN {X 0,Y 470.141,Z 686.468,A -85,B 0,C 180,E1 22162.376,E2 22162.376} C_VEL
LIN {X 0,Y 468.055,Z 682.703,A -85,B 0,C 180,E1 22161.557,E2 22161.557} C_VEL
LIN {X 0,Y 467.099,Z 681.275,A -85,B 0,C 180,E1 22161.208,E2 22161.208} C_VEL
LIN {X 0,Y 465.307,Z 678.22,A -85,B 0,C 180,E1 22160.503,E2 22160.503} C_VEL
LIN {X 0,Y 465.004,Z 676.81,A -85,B 0,C 180,E1 22160.254,E2 22160.254} C_VEL
LIN {X 0,Y 465.014,Z 676.814,A -85,B 0,C 180,E1 22156.488,E2 22156.488} C_VEL
LIN {X 0,Y 465,Z 676.814,A -85,B 0,C 180,E1 22152.922,E2 22152.922} C_VEL
LIN {X 0,Y 465.011,Z 676.813,A -85,B 0,C 180,E1 22149.278,E2 22149.278} C_VEL
LIN {X 0,Y 465.013,Z 676.813,A -85,B 0,C 180,E1 22145.676,E2 22145.676} C_VEL
LIN {X 0,Y 465.002,Z 676.812,A -85,B 0,C 180,E1 22141.971,E2 22141.971} C_VEL
LIN {X 0,Y 465.015,Z 676.81,A -85,B 0,C 180,E1 22138.275,E2 22138.275} C_VEL
LIN {X 0,Y 465.008,Z 676.812,A -85,B 0,C 180,E1 22134.571,E2 22134.571} C_VEL
LIN {X 0,Y 465.011,Z 676.81,A -85,B 0,C 180,E1 22130.844,E2 22130.844} C_VEL
LIN {X 0,Y 465.01,Z 676.811,A -85,B 0,C 180,E1 22127.204,E2 22127.204} C_VEL
LIN {X 0,Y 465.01,Z 676.811,A -85,B 0,C 180,E1 22123.53,E2 22123.53} C_VEL
LIN {X 0,Y 465.011,Z 676.807,A -85,B 0,C 180,E1 22119.746,E2 22119.746} C_VEL
LIN {X 0,Y 465.005,Z 676.806,A -85,B 0,C 180,E1 22116.156,E2 22116.156} C_VEL
LIN {X 0,Y 465.013,Z 676.784,A -85,B 0,C 180,E1 22112.465,E2 22112.465} C_VEL
LIN {X 0,Y 465.017,Z 676.804,A -85,B 0,C 180,E1 22108.789,E2 22108.789} C_VEL
LIN {X 0,Y 465.006,Z 676.779,A -85,B 0,C 180,E1 22105.113,E2 22105.113} C_VEL
LIN {X 0,Y 465.016,Z 676.81,A -85,B 0,C 180,E1 22101.306,E2 22101.306} C_VEL
LIN {X 0,Y 465.015,Z 676.803,A -85,B 0,C 180,E1 22097.518,E2 22097.518} C_VEL
LIN {X 0,Y 465.034,Z 676.963,A -85,B 0,C 180,E1 22094.995,E2 22094.995} C_VEL
LIN {X 0,Y 466.219,Z 680.158,A -85,B 0,C 180,E1 22094.601,E2 22094.601} C_VEL
LIN {X 0,Y 467.549,Z 682.763,A -85,B 0,C 180,E1 22094.242,E2 22094.242} C_VEL
LIN {X 0,Y 474.858,Z 698.207,A -85,B 0,C 180,E1 22092.169,E2 22092.169} C_VEL
LIN {X 0,Y 483.816,Z 719.436,A -85,B 0,C 180,E1 22089.532,E2 22089.532} C_VEL
LIN {X 0,Y 483.929,Z 722.283,A -85,B 0,C 180,E1 22089.291,E2 22089.291} C_VEL
LIN {X 0,Y 481.941,Z 765.076,A -85,B 0,C 180,E1 22086.192,E2 22086.192} C_VEL
LIN {X 0,Y 481.927,Z 771.167,A -85,B 0,C 180,E1 22085.812,E2 22085.812} C_VEL
LIN {X 0,Y 484.601,Z 789.708,A -85,B 0,C 180,E1 22085.248,E2 22085.248} C_VEL
LIN {X 0,Y 484.245,Z 808.717,A -85,B 0,C 180,E1 22084.938,E2 22084.938} C_VEL
LIN {X 0,Y 483.276,Z 816.411,A -85,B 0,C 180,E1 22084.882,E2 22084.882} C_VEL
LIN {X 0,Y 477.759,Z 836.922,A -85,B 0,C 180,E1 22084.979,E2 22084.979} C_VEL
LIN {X 0,Y 477.036,Z 843.523,A -85,B 0,C 180,E1 22084.921,E2 22084.921} C_VEL
LIN {X 0,Y 473.376,Z 1032.163,A -85,B 0,C 180,E1 22081.81,E2 22081.81} C_VEL
LIN {X 0,Y 472.516,Z 1053.02,A -85,B 0,C 180,E1 22081.254,E2 22081.254} C_VEL
LIN {X 0,Y 471.328,Z 1073.601,A -85,B 0,C 180,E1 22080.464,E2 22080.464} C_VEL
LIN {X 0,Y 469.89,Z 1092.631,A -85,B 0,C 180,E1 22079.507,E2 22079.507} C_VEL
LIN {X 0,Y 468.301,Z 1110.809,A -85,B 0,C 180,E1 22078.362,E2 22078.362} C_VEL
LIN {X 0,Y 466.477,Z 1128.988,A -85,B 0,C 180,E1 22076.957,E2 22076.957} C_VEL
LIN {X 0,Y 464.609,Z 1146.061,A -85,B 0,C 180,E1 22075.356,E2 22075.356} C_VEL
LIN {X 0,Y 462.851,Z 1161.243,A -85,B 0,C 180,E1 22073.661,E2 22073.661} C_VEL
LIN {X 0,Y 461.187,Z 1175.658,A -85,B 0,C 180,E1 22071.76,E2 22071.76} C_VEL
LIN {X 0,Y 459.667,Z 1189.235,A -85,B 0,C 180,E1 22069.634,E2 22069.634} C_VEL
LIN {X 0,Y 458.48,Z 1200.651,A -85,B 0,C 180,E1 22067.514,E2 22067.514} C_VEL
LIN {X 0,Y 457.51,Z 1211.049,A -85,B 0,C 180,E1 22065.203,E2 22065.203} C_VEL
LIN {X 0,Y 456.766,Z 1220.402,A -85,B 0,C 180,E1 22062.644,E2 22062.644} C_VEL
LIN {X 0,Y 456.316,Z 1227.746,A -85,B 0,C 180,E1 22060.095,E2 22060.095} C_VEL
LIN {X 0,Y 456.074,Z 1233.292,A -85,B 0,C 180,E1 22057.558,E2 22057.558} C_VEL
LIN {X 0,Y 455.971,Z 1237.182,A -85,B 0,C 180,E1 22055.031,E2 22055.031} C_VEL
LIN {X 0,Y 455.942,Z 1239.519,A -85,B 0,C 180,E1 22052.513,E2 22052.513} C_VEL
LIN {X 0,Y 455.941,Z 1240.338,A -85,B 0,C 180,E1 22049.999,E2 22049.999} C_VEL
LIN {X 0,Y 455.94,Z 1239.501,A -85,B 0,C 180,E1 22047.36,E2 22047.36} C_VEL
LIN {X 0,Y 455.973,Z 1237.14,A -85,B 0,C 180,E1 22044.841,E2 22044.841} C_VEL
LIN {X 0,Y 456.093,Z 1232.975,A -85,B 0,C 180,E1 22042.188,E2 22042.188} C_VEL
LIN {X 0,Y 456.334,Z 1227.302,A -85,B 0,C 180,E1 22039.649,E2 22039.649} C_VEL
LIN {X 0,Y 456.777,Z 1220.264,A -85,B 0,C 180,E1 22037.227,E2 22037.227} C_VEL
LIN {X 0,Y 457.478,Z 1211.402,A -85,B 0,C 180,E1 22034.795,E2 22034.795} C_VEL
LIN {X 0,Y 458.502,Z 1200.454,A -85,B 0,C 180,E1 22032.355,E2 22032.355} C_VEL
LIN {X 0,Y 459.739,Z 1188.607,A -85,B 0,C 180,E1 22030.167,E2 22030.167} C_VEL
LIN {X 0,Y 461.233,Z 1175.294,A -85,B 0,C 180,E1 22028.098,E2 22028.098} C_VEL
LIN {X 0,Y 462.978,Z 1160.111,A -85,B 0,C 180,E1 22026.113,E2 22026.113} C_VEL
LIN {X 0,Y 464.858,Z 1143.712,A -85,B 0,C 180,E1 22024.32,E2 22024.32} C_VEL
LIN {X 0,Y 466.713,Z 1126.595,A -85,B 0,C 180,E1 22022.757,E2 22022.757} C_VEL
LIN {X 0,Y 468.45,Z 1109.218,A -85,B 0,C 180,E1 22021.438,E2 22021.438} C_VEL
LIN {X 0,Y 470.073,Z 1090.691,A -85,B 0,C 180,E1 22020.29,E2 22020.29} C_VEL
LIN {X 0,Y 471.497,Z 1071.133,A -85,B 0,C 180,E1 22019.335,E2 22019.335} C_VEL
LIN {X 0,Y 472.604,Z 1051.325,A -85,B 0,C 180,E1 22018.602,E2 22018.602} C_VEL
LIN {X 0,Y 473.421,Z 1030.515,A -85,B 0,C 180,E1 22018.065,E2 22018.065} C_VEL
LIN {X 0,Y 477.96,Z 797.519,A -85,B 0,C 180,E1 22014.23,E2 22014.23} C_VEL
LIN {X 0,Y 472.376,Z 772.523,A -85,B 0,C 180,E1 22013.238,E2 22013.238} C_VEL
LIN {X 0,Y 473.571,Z 745.222,A -85,B 0,C 180,E1 22010.456,E2 22010.456} C_VEL
LIN {X 0,Y 474.894,Z 723.708,A -85,B 0,C 180,E1 22008.131,E2 22008.131} C_VEL
LIN {X 0,Y 468.312,Z 704.995,A -85,B 0,C 180,E1 22005.206,E2 22005.206} C_VEL
LIN {X 0,Y 462.074,Z 689.371,A -85,B 0,C 180,E1 22002.632,E2 22002.632} C_VEL
LIN {X 0,Y 460.257,Z 685.368,A -85,B 0,C 180,E1 22001.914,E2 22001.914} C_VEL
LIN {X 0,Y 467.571,Z 702.344,A -85,B 0,C 180,E1 21999.179,E2 21999.179} C_VEL
LIN {X 0,Y 474.384,Z 719.746,A -85,B 0,C 180,E1 21996.579,E2 21996.579} C_VEL
LIN {X 0,Y 475.463,Z 722.833,A -85,B 0,C 180,E1 21996.145,E2 21996.145} C_VEL
LIN {X 0,Y 472.438,Z 761.467,A -85,B 0,C 180,E1 21992.446,E2 21992.446} C_VEL
LIN {X 0,Y 469.465,Z 802.72,A -85,B 0,C 180,E1 21988.564,E2 21988.564} C_VEL
LIN {X 0,Y 466.749,Z 844.548,A -85,B 0,C 180,E1 21984.691,E2 21984.691} C_VEL
LIN {X 0,Y 466.273,Z 854.763,A -85,B 0,C 180,E1 21983.788,E2 21983.788} C_VEL
LIN {X 0,Y 467.491,Z 864.546,A -85,B 0,C 180,E1 21983.513,E2 21983.513} C_VEL
LIN {X 0,Y 464.107,Z 1025.135,A -85,B 0,C 180,E1 21980.583,E2 21980.583} C_VEL
LIN {X 0,Y 463.617,Z 1042.961,A -85,B 0,C 180,E1 21980.013,E2 21980.013} C_VEL
LIN {X 0,Y 462.921,Z 1059.948,A -85,B 0,C 180,E1 21979.232,E2 21979.232} C_VEL
LIN {X 0,Y 462.094,Z 1075.386,A -85,B 0,C 180,E1 21978.285,E2 21978.285} C_VEL
LIN {X 0,Y 461.115,Z 1090.693,A -85,B 0,C 180,E1 21977.087,E2 21977.087} C_VEL
LIN {X 0,Y 460.15,Z 1104.707,A -85,B 0,C 180,E1 21975.72,E2 21975.72} C_VEL
LIN {X 0,Y 459.248,Z 1117.088,A -85,B 0,C 180,E1 21974.242,E2 21974.242} C_VEL
LIN {X 0,Y 458.432,Z 1128.351,A -85,B 0,C 180,E1 21972.598,E2 21972.598} C_VEL
LIN {X 0,Y 457.727,Z 1138.205,A -85,B 0,C 180,E1 21970.828,E2 21970.828} C_VEL
LIN {X 0,Y 457.149,Z 1147.207,A -85,B 0,C 180,E1 21968.807,E2 21968.807} C_VEL
LIN {X 0,Y 456.806,Z 1154.201,A -85,B 0,C 180,E1 21966.788,E2 21966.788} C_VEL
LIN {X 0,Y 456.575,Z 1159.683,A -85,B 0,C 180,E1 21964.648,E2 21964.648} C_VEL
LIN {X 0,Y 456.463,Z 1163.362,A -85,B 0,C 180,E1 21962.511,E2 21962.511} C_VEL
LIN {X 0,Y 456.442,Z 1165.472,A -85,B 0,C 180,E1 21960.251,E2 21960.251} C_VEL
LIN {X 0,Y 456.455,Z 1165.85,A -85,B 0,C 180,E1 21958.117,E2 21958.117} C_VEL
LIN {X 0,Y 456.545,Z 1164.598,A -85,B 0,C 180,E1 21955.982,E2 21955.982} C_VEL
LIN {X 0,Y 456.689,Z 1161.704,A -85,B 0,C 180,E1 21953.842,E2 21953.842} C_VEL
LIN {X 0,Y 456.957,Z 1157.11,A -85,B 0,C 180,E1 21951.697,E2 21951.697} C_VEL
LIN {X 0,Y 457.362,Z 1151.032,A -85,B 0,C 180,E1 21949.662,E2 21949.662} C_VEL
LIN {X 0,Y 457.94,Z 1143.043,A -85,B 0,C 180,E1 21947.645,E2 21947.645} C_VEL
LIN {X 0,Y 458.731,Z 1133.446,A -85,B 0,C 180,E1 21945.742,E2 21945.742} C_VEL
LIN {X 0,Y 459.601,Z 1122.964,A -85,B 0,C 180,E1 21944.065,E2 21944.065} C_VEL
LIN {X 0,Y 460.545,Z 1110.869,A -85,B 0,C 180,E1 21942.501,E2 21942.501} C_VEL
LIN {X 0,Y 461.532,Z 1097.503,A -85,B 0,C 180,E1 21941.103,E2 21941.103} C_VEL
LIN {X 0,Y 462.475,Z 1083.129,A -85,B 0,C 180,E1 21939.895,E2 21939.895} C_VEL
LIN {X 0,Y 463.219,Z 1068.744,A -85,B 0,C 180,E1 21938.938,E2 21938.938} C_VEL
LIN {X 0,Y 463.822,Z 1052.821,A -85,B 0,C 180,E1 21938.137,E2 21938.137} C_VEL
LIN {X 0,Y 464.213,Z 1035.587,A -85,B 0,C 180,E1 21937.523,E2 21937.523} C_VEL
LIN {X 0,Y 464.801,Z 1002.807,A -85,B 0,C 180,E1 21936.809,E2 21936.809} C_VEL
LIN {X 0,Y 467.647,Z 927.969,A -85,B 0,C 180,E1 21935.166,E2 21935.166} C_VEL
LIN {X 0,Y 470.376,Z 877.218,A -85,B 0,C 180,E1 21933.963,E2 21933.963} C_VEL
LIN {X 0,Y 474.517,Z 866.655,A -85,B 0,C 180,E1 21933.198,E2 21933.198} C_VEL
LIN {X 0,Y 480.309,Z 838.125,A -85,B 0,C 180,E1 21929.957,E2 21929.957} C_VEL
LIN {X 0,Y 486.67,Z 816.365,A -85,B 0,C 180,E1 21927.294,E2 21927.294} C_VEL
LIN {X 0,Y 493.349,Z 800.232,A -85,B 0,C 180,E1 21925.144,E2 21925.144} C_VEL
LIN {X 0,Y 497.139,Z 793.201,A -85,B 0,C 180,E1 21924.147,E2 21924.147} C_VEL
LIN {X 0,Y 490.703,Z 802.985,A -85,B 0,C 180,E1 21922.817,E2 21922.817} C_VEL
LIN {X 0,Y 486.609,Z 812.522,A -85,B 0,C 180,E1 21921.495,E2 21921.495} C_VEL
LIN {X 0,Y 484.712,Z 822.133,A -85,B 0,C 180,E1 21920.164,E2 21920.164} C_VEL
LIN {X 0,Y 484.962,Z 832.148,A -85,B 0,C 180,E1 21918.81,E2 21918.81} C_VEL
LIN {X 0,Y 487.202,Z 841.875,A -85,B 0,C 180,E1 21917.532,E2 21917.532} C_VEL
LIN {X 0,Y 491.635,Z 852.079,A -85,B 0,C 180,E1 21916.218,E2 21916.218} C_VEL
LIN {X 0,Y 498.401,Z 862.362,A -85,B 0,C 180,E1 21914.915,E2 21914.915} C_VEL
LIN {X 0,Y 507.356,Z 872.252,A -85,B 0,C 180,E1 21913.677,E2 21913.677} C_VEL
LIN {X 0,Y 518.316,Z 881.306,A -85,B 0,C 180,E1 21912.533,E2 21912.533} C_VEL
LIN {X 0,Y 530.446,Z 888.973,A -85,B 0,C 180,E1 21911.555,E2 21911.555} C_VEL
LIN {X 0,Y 538.665,Z 893.281,A -85,B 0,C 180,E1 21911.001,E2 21911.001} C_VEL
LIN {X 0,Y 514.396,Z 929.297,A -85,B 0,C 180,E1 21910.045,E2 21910.045} C_VEL
LIN {X 0,Y 503.521,Z 948.227,A -85,B 0,C 180,E1 21909.453,E2 21909.453} C_VEL
LIN {X 0,Y 496.312,Z 963.947,A -85,B 0,C 180,E1 21908.869,E2 21908.869} C_VEL
LIN {X 0,Y 493.97,Z 969.666,A -85,B 0,C 180,E1 21908.642,E2 21908.642} C_VEL
LIN {X 0,Y 486.595,Z 985.232,A -85,B 0,C 180,E1 21908.057,E2 21908.057} C_VEL
LIN {X 0,Y 477.366,Z 1011.958,A -85,B 0,C 180,E1 21906.876,E2 21906.876} C_VEL
LIN {X 0,Y 476.7,Z 1015.022,A -85,B 0,C 180,E1 21906.774,E2 21906.774} C_VEL
LIN {X 0,Y 475.448,Z 1027.551,A -85,B 0,C 180,E1 21906.632,E2 21906.632} C_VEL
LIN {X 0,Y 474.754,Z 1061.164,A -85,B 0,C 180,E1 21906.043,E2 21906.043} C_VEL
LIN {X 0,Y 473.666,Z 1085.578,A -85,B 0,C 180,E1 21905.399,E2 21905.399} C_VEL
LIN {X 0,Y 472.351,Z 1108.745,A -85,B 0,C 180,E1 21904.562,E2 21904.562} C_VEL
LIN {X 0,Y 470.847,Z 1132.45,A -85,B 0,C 180,E1 21903.465,E2 21903.465} C_VEL
LIN {X 0,Y 469.175,Z 1154.558,A -85,B 0,C 180,E1 21902.194,E2 21902.194} C_VEL
LIN {X 0,Y 467.42,Z 1176.03,A -85,B 0,C 180,E1 21900.693,E2 21900.693} C_VEL
LIN {X 0,Y 465.656,Z 1195.975,A -85,B 0,C 180,E1 21899.03,E2 21899.03} C_VEL
LIN {X 0,Y 463.762,Z 1215.703,A -85,B 0,C 180,E1 21897.075,E2 21897.075} C_VEL
LIN {X 0,Y 462.178,Z 1231.452,A -85,B 0,C 180,E1 21895.226,E2 21895.226} C_VEL
LIN {X 0,Y 461.209,Z 1241.221,A -85,B 0,C 180,E1 21893.917,E2 21893.917} C_VEL
LIN {X 0,Y 460.119,Z 1251.044,A -85,B 0,C 180,E1 21892.352,E2 21892.352} C_VEL
LIN {X 0,Y 458.894,Z 1262.211,A -85,B 0,C 180,E1 21890.27,E2 21890.27} C_VEL
LIN {X 0,Y 457.93,Z 1271.92,A -85,B 0,C 180,E1 21888.194,E2 21888.194} C_VEL
LIN {X 0,Y 457.065,Z 1282.277,A -85,B 0,C 180,E1 21885.609,E2 21885.609} C_VEL
LIN {X 0,Y 456.496,Z 1290.609,A -85,B 0,C 180,E1 21883.039,E2 21883.039} C_VEL
LIN {X 0,Y 456.186,Z 1296.74,A -85,B 0,C 180,E1 21880.737,E2 21880.737} C_VEL
LIN {X 0,Y 456.008,Z 1302.128,A -85,B 0,C 180,E1 21878.194,E2 21878.194} C_VEL
LIN {X 0,Y 455.929,Z 1306.302,A -85,B 0,C 180,E1 21875.363,E2 21875.363} C_VEL
LIN {X 0,Y 455.903,Z 1308.508,A -85,B 0,C 180,E1 21872.892,E2 21872.892} C_VEL
LIN {X 0,Y 455.896,Z 1309.41,A -85,B 0,C 180,E1 21870.503,E2 21870.503} C_VEL
LIN {X 0,Y 455.905,Z 1308.839,A -85,B 0,C 180,E1 21867.612,E2 21867.612} C_VEL
LIN {X 0,Y 455.917,Z 1306.796,A -85,B 0,C 180,E1 21865.094,E2 21865.094} C_VEL
LIN {X 0,Y 455.97,Z 1303.592,A -85,B 0,C 180,E1 21862.694,E2 21862.694} C_VEL
LIN {X 0,Y 456.129,Z 1298.595,A -85,B 0,C 180,E1 21860.028,E2 21860.028} C_VEL
LIN {X 0,Y 456.442,Z 1291.73,A -85,B 0,C 180,E1 21857.347,E2 21857.347} C_VEL
LIN {X 0,Y 456.902,Z 1284.461,A -85,B 0,C 180,E1 21855.036,E2 21855.036} C_VEL
LIN {X 0,Y 457.697,Z 1274.769,A -85,B 0,C 180,E1 21852.455,E2 21852.455} C_VEL
LIN {X 0,Y 458.788,Z 1263.23,A -85,B 0,C 180,E1 21849.933,E2 21849.933} C_VEL
LIN {X 0,Y 459.948,Z 1252.512,A -85,B 0,C 180,E1 21847.91,E2 21847.91} C_VEL
LIN {X 0,Y 460.923,Z 1243.84,A -85,B 0,C 180,E1 21846.476,E2 21846.476} C_VEL
LIN {X 0,Y 462.2,Z 1231.746,A -85,B 0,C 180,E1 21844.777,E2 21844.777} C_VEL
LIN {X 0,Y 463.832,Z 1216.636,A -85,B 0,C 180,E1 21842.908,E2 21842.908} C_VEL
LIN {X 0,Y 465.948,Z 1197.146,A -85,B 0,C 180,E1 21840.85,E2 21840.85} C_VEL
LIN {X 0,Y 468.026,Z 1177.419,A -85,B 0,C 180,E1 21839.084,E2 21839.084} C_VEL
LIN {X 0,Y 470.095,Z 1156.603,A -85,B 0,C 180,E1 21837.518,E2 21837.518} C_VEL
LIN {X 0,Y 472.107,Z 1135.526,A -85,B 0,C 180,E1 21836.204,E2 21836.204} C_VEL
LIN {X 0,Y 473.936,Z 1113.538,A -85,B 0,C 180,E1 21835.087,E2 21835.087} C_VEL
LIN {X 0,Y 475.659,Z 1090.113,A -85,B 0,C 180,E1 21834.161,E2 21834.161} C_VEL
LIN {X 0,Y 476.97,Z 1068.132,A -85,B 0,C 180,E1 21833.521,E2 21833.521} C_VEL
LIN {X 0,Y 477.844,Z 1043.503,A -85,B 0,C 180,E1 21833.033,E2 21833.033} C_VEL
LIN {X 0,Y 478.657,Z 1020.636,A -85,B 0,C 180,E1 21832.662,E2 21832.662} C_VEL
LIN {X 0,Y 483.469,Z 1005.269,A -85,B 0,C 180,E1 21831.955,E2 21831.955} C_VEL
LIN {X 0,Y 490.691,Z 985.98,A -85,B 0,C 180,E1 21831.128,E2 21831.128} C_VEL
LIN {X 0,Y 498.191,Z 969.974,A -85,B 0,C 180,E1 21830.581,E2 21830.581} C_VEL
LIN {X 0,Y 504.475,Z 955.115,A -85,B 0,C 180,E1 21830.048,E2 21830.048} C_VEL
LIN {X 0,Y 513.962,Z 936.976,A -85,B 0,C 180,E1 21829.551,E2 21829.551} C_VEL
LIN {X 0,Y 531.038,Z 908.78,A -85,B 0,C 180,E1 21828.985,E2 21828.985} C_VEL
LIN {X 0,Y 540.026,Z 894.518,A -85,B 0,C 180,E1 21828.738,E2 21828.738} C_VEL
LIN {X 0,Y 528.089,Z 888.857,A -85,B 0,C 180,E1 21827.435,E2 21827.435} C_VEL
LIN {X 0,Y 517.869,Z 881.818,A -85,B 0,C 180,E1 21826.067,E2 21826.067} C_VEL
LIN {X 0,Y 509.759,Z 874.056,A -85,B 0,C 180,E1 21824.761,E2 21824.761} C_VEL
LIN {X 0,Y 502.108,Z 863.765,A -85,B 0,C 180,E1 21823.236,E2 21823.236} C_VEL
LIN {X 0,Y 496.159,Z 851.794,A -85,B 0,C 180,E1 21821.683,E2 21821.683} C_VEL
LIN {X 0,Y 492.18,Z 839.218,A -85,B 0,C 180,E1 21820.241,E2 21820.241} C_VEL
LIN {X 0,Y 489.692,Z 824.645,A -85,B 0,C 180,E1 21818.743,E2 21818.743} C_VEL
LIN {X 0,Y 488.834,Z 808.434,A -85,B 0,C 180,E1 21817.26,E2 21817.26} C_VEL
LIN {X 0,Y 489.853,Z 788.234,A -85,B 0,C 180,E1 21815.615,E2 21815.615} C_VEL
LIN {X 0,Y 493.939,Z 747.41,A -85,B 0,C 180,E1 21812.44,E2 21812.44} C_VEL
LIN {X 0,Y 493.951,Z 744.902,A -85,B 0,C 180,E1 21812.21,E2 21812.21} C_VEL
LIN {X 0,Y 483.922,Z 725.97,A -85,B 0,C 180,E1 21808.913,E2 21808.913} C_VEL
LIN {X 0,Y 475.624,Z 711.098,A -85,B 0,C 180,E1 21806.063,E2 21806.063} C_VEL
LIN {X 0,Y 470.182,Z 701.509,A -85,B 0,C 180,E1 21804.097,E2 21804.097} C_VEL
LIN {X 0,Y 467.724,Z 697.135,A -85,B 0,C 180,E1 21803.162,E2 21803.162} C_VEL
LIN {X 0,Y 464.942,Z 692.281,A -85,B 0,C 180,E1 21802.107,E2 21802.107} C_VEL
LIN {X 0,Y 462.266,Z 687.519,A -85,B 0,C 180,E1 21801.042,E2 21801.042} C_VEL
LIN {X 0,Y 460.176,Z 683.885,A -85,B 0,C 180,E1 21800.21,E2 21800.21} C_VEL
LIN {X 0,Y 459.648,Z 682.745,A -85,B 0,C 180,E1 21799.969,E2 21799.969} C_VEL
LIN {X 0,Y 457.713,Z 680.106,A -85,B 0,C 180,E1 21799.26,E2 21799.26} C_VEL
LIN {X 0,Y 457.07,Z 677.798,A -85,B 0,C 180,E1 21798.824,E2 21798.824} C_VEL
LIN {X 0,Y 457.081,Z 677.799,A -85,B 0,C 180,E1 21795.088,E2 21795.088} C_VEL
LIN {X 0,Y 457.074,Z 677.801,A -85,B 0,C 180,E1 21791.226,E2 21791.226} C_VEL
LIN {X 0,Y 457.065,Z 677.802,A -85,B 0,C 180,E1 21787.542,E2 21787.542} C_VEL
LIN {X 0,Y 457.073,Z 677.801,A -85,B 0,C 180,E1 21783.888,E2 21783.888} C_VEL
LIN {X 0,Y 457.068,Z 677.797,A -85,B 0,C 180,E1 21780.125,E2 21780.125} C_VEL
LIN {X 0,Y 457.073,Z 677.799,A -85,B 0,C 180,E1 21776.488,E2 21776.488} C_VEL
LIN {X 0,Y 457.065,Z 677.802,A -85,B 0,C 180,E1 21772.71,E2 21772.71} C_VEL
LIN {X 0,Y 457.069,Z 677.799,A -85,B 0,C 180,E1 21769.028,E2 21769.028} C_VEL
LIN {X 0,Y 457.072,Z 677.801,A -85,B 0,C 180,E1 21765.3,E2 21765.3} C_VEL
LIN {X 0,Y 457.062,Z 677.797,A -85,B 0,C 180,E1 21761.638,E2 21761.638} C_VEL
LIN {X 0,Y 457.078,Z 677.797,A -85,B 0,C 180,E1 21757.898,E2 21757.898} C_VEL
LIN {X 0,Y 457.063,Z 677.801,A -85,B 0,C 180,E1 21754.194,E2 21754.194} C_VEL
LIN {X 0,Y 457.067,Z 677.758,A -85,B 0,C 180,E1 21750.514,E2 21750.514} C_VEL
LIN {X 0,Y 457.066,Z 677.797,A -85,B 0,C 180,E1 21746.846,E2 21746.846} C_VEL
LIN {X 0,Y 457.062,Z 677.781,A -85,B 0,C 180,E1 21743.173,E2 21743.173} C_VEL
LIN {X 0,Y 457.073,Z 677.769,A -85,B 0,C 180,E1 21739.574,E2 21739.574} C_VEL
LIN {X 0,Y 457.067,Z 677.835,A -85,B 0,C 180,E1 21735.863,E2 21735.863} C_VEL
LIN {X 0,Y 458.019,Z 680.711,A -85,B 0,C 180,E1 21735.513,E2 21735.513} C_VEL
LIN {X 0,Y 459.402,Z 683.063,A -85,B 0,C 180,E1 21735.157,E2 21735.157} C_VEL
LIN {X 0,Y 467.904,Z 700.956,A -85,B 0,C 180,E1 21732.685,E2 21732.685} C_VEL
LIN {X 0,Y 476.711,Z 721.8,A -85,B 0,C 180,E1 21730.043,E2 21730.043} C_VEL
LIN {X 0,Y 477.348,Z 724.203,A -85,B 0,C 180,E1 21729.784,E2 21729.784} C_VEL
LIN {X 0,Y 475.332,Z 766.167,A -85,B 0,C 180,E1 21726.733,E2 21726.733} C_VEL
LIN {X 0,Y 475.311,Z 771.611,A -85,B 0,C 180,E1 21726.39,E2 21726.39} C_VEL
LIN {X 0,Y 478.088,Z 790.915,A -85,B 0,C 180,E1 21725.788,E2 21725.788} C_VEL
LIN {X 0,Y 477.036,Z 843.523,A -85,B 0,C 180,E1 21724.921,E2 21724.921} C_VEL
LIN {X 0,Y 476.092,Z 851.212,A -85,B 0,C 180,E1 21724.862,E2 21724.862} C_VEL
LIN {X 0,Y 470.539,Z 871.71,A -85,B 0,C 180,E1 21724.964,E2 21724.964} C_VEL
LIN {X 0,Y 469.775,Z 878.313,A -85,B 0,C 180,E1 21724.909,E2 21724.909} C_VEL
LIN {X 0,Y 466.604,Z 1032.853,A -85,B 0,C 180,E1 21722.323,E2 21722.323} C_VEL
LIN {X 0,Y 465.705,Z 1053.629,A -85,B 0,C 180,E1 21721.761,E2 21721.761} C_VEL
LIN {X 0,Y 464.457,Z 1074.166,A -85,B 0,C 180,E1 21720.964,E2 21720.964} C_VEL
LIN {X 0,Y 462.942,Z 1093.221,A -85,B 0,C 180,E1 21719.994,E2 21719.994} C_VEL
LIN {X 0,Y 461.26,Z 1111.396,A -85,B 0,C 180,E1 21718.835,E2 21718.835} C_VEL
LIN {X 0,Y 459.33,Z 1129.578,A -85,B 0,C 180,E1 21717.411,E2 21717.411} C_VEL
LIN {X 0,Y 457.344,Z 1146.656,A -85,B 0,C 180,E1 21715.788,E2 21715.788} C_VEL
LIN {X 0,Y 455.437,Z 1162.102,A -85,B 0,C 180,E1 21714.037,E2 21714.037} C_VEL
LIN {X 0,Y 453.695,Z 1176.262,A -85,B 0,C 180,E1 21712.138,E2 21712.138} C_VEL
LIN {X 0,Y 452.108,Z 1189.46,A -85,B 0,C 180,E1 21710.046,E2 21710.046} C_VEL
LIN {X 0,Y 450.774,Z 1201.263,A -85,B 0,C 180,E1 21707.823,E2 21707.823} C_VEL
LIN {X 0,Y 449.717,Z 1211.663,A -85,B 0,C 180,E1 21705.473,E2 21705.473} C_VEL
LIN {X 0,Y 448.902,Z 1221.016,A -85,B 0,C 180,E1 21702.869,E2 21702.869} C_VEL
LIN {X 0,Y 448.399,Z 1228.359,A -85,B 0,C 180,E1 21700.275,E2 21700.275} C_VEL
LIN {X 0,Y 448.129,Z 1233.904,A -85,B 0,C 180,E1 21697.693,E2 21697.693} C_VEL
LIN {X 0,Y 448.003,Z 1237.793,A -85,B 0,C 180,E1 21695.121,E2 21695.121} C_VEL
LIN {X 0,Y 447.967,Z 1240.128,A -85,B 0,C 180,E1 21692.558,E2 21692.558} C_VEL
LIN {X 0,Y 447.964,Z 1240.947,A -85,B 0,C 180,E1 21689.999,E2 21689.999} C_VEL
LIN {X 0,Y 447.966,Z 1240.11,A -85,B 0,C 180,E1 21687.313,E2 21687.313} C_VEL
LIN {X 0,Y 448.006,Z 1237.749,A -85,B 0,C 180,E1 21684.749,E2 21684.749} C_VEL
LIN {X 0,Y 448.147,Z 1233.584,A -85,B 0,C 180,E1 21682.048,E2 21682.048} C_VEL
LIN {X 0,Y 448.419,Z 1227.912,A -85,B 0,C 180,E1 21679.464,E2 21679.464} C_VEL
LIN {X 0,Y 448.914,Z 1220.873,A -85,B 0,C 180,E1 21676.999,E2 21676.999} C_VEL
LIN {X 0,Y 449.683,Z 1212.01,A -85,B 0,C 180,E1 21674.525,E2 21674.525} C_VEL
LIN {X 0,Y 450.767,Z 1201.313,A -85,B 0,C 180,E1 21672.097,E2 21672.097} C_VEL
LIN {X 0,Y 452.044,Z 1189.949,A -85,B 0,C 180,E1 21669.95,E2 21669.95} C_VEL
LIN {X 0,Y 453.622,Z 1176.848,A -85,B 0,C 180,E1 21667.857,E2 21667.857} C_VEL
LIN {X 0,Y 455.415,Z 1162.307,A -85,B 0,C 180,E1 21665.898,E2 21665.898} C_VEL
LIN {X 0,Y 457.31,Z 1146.981,A -85,B 0,C 180,E1 21664.154,E2 21664.154} C_VEL
LIN {X 0,Y 459.309,Z 1129.791,A -85,B 0,C 180,E1 21662.516,E2 21662.516} C_VEL
LIN {X 0,Y 461.24,Z 1111.633,A -85,B 0,C 180,E1 21661.091,E2 21661.091} C_VEL
LIN {X 0,Y 462.926,Z 1093.433,A -85,B 0,C 180,E1 21659.927,E2 21659.927} C_VEL
LIN {X 0,Y 464.436,Z 1074.551,A -85,B 0,C 180,E1 21658.963,E2 21658.963} C_VEL
LIN {X 0,Y 465.685,Z 1054.063,A -85,B 0,C 180,E1 21658.162,E2 21658.162} C_VEL
LIN {X 0,Y 466.584,Z 1033.628,A -85,B 0,C 180,E1 21657.602,E2 21657.602} C_VEL
LIN {X 0,Y 468.107,Z 960.774,A -85,B 0,C 180,E1 21656.366,E2 21656.366} C_VEL
LIN {X 0,Y 471.344,Z 798.144,A -85,B 0,C 180,E1 21653.652,E2 21653.652} C_VEL
LIN {X 0,Y 465.674,Z 773.375,A -85,B 0,C 180,E1 21652.653,E2 21652.653} C_VEL
LIN {X 0,Y 466.919,Z 746.155,A -85,B 0,C 180,E1 21649.861,E2 21649.861} C_VEL
LIN {X 0,Y 467.99,Z 726.808,A -85,B 0,C 180,E1 21647.748,E2 21647.748} C_VEL
LIN {X 0,Y 461.405,Z 708.118,A -85,B 0,C 180,E1 21644.771,E2 21644.771} C_VEL
LIN {X 0,Y 455.482,Z 693.436,A -85,B 0,C 180,E1 21642.288,E2 21642.288} C_VEL
LIN {X 0,Y 454.611,Z 691.481,A -85,B 0,C 180,E1 21641.915,E2 21641.915} C_VEL
LIN {X 0,Y 461.988,Z 708.714,A -85,B 0,C 180,E1 21639.114,E2 21639.114} C_VEL
LIN {X 0,Y 468.66,Z 726.212,A -85,B 0,C 180,E1 21636.488,E2 21636.488} C_VEL
LIN {X 0,Y 465.525,Z 764.824,A -85,B 0,C 180,E1 21632.769,E2 21632.769} C_VEL
LIN {X 0,Y 462.374,Z 806.286,A -85,B 0,C 180,E1 21628.831,E2 21628.831} C_VEL
LIN {X 0,Y 459.548,Z 847.623,A -85,B 0,C 180,E1 21624.967,E2 21624.967} C_VEL
LIN {X 0,Y 459.151,Z 855.749,A -85,B 0,C 180,E1 21624.242,E2 21624.242} C_VEL
LIN {X 0,Y 460.392,Z 865.476,A -85,B 0,C 180,E1 21623.959,E2 21623.959} C_VEL
LIN {X 0,Y 456.689,Z 1026.276,A -85,B 0,C 180,E1 21620.939,E2 21620.939} C_VEL
LIN {X 0,Y 456.178,Z 1044.062,A -85,B 0,C 180,E1 21620.358,E2 21620.358} C_VEL
LIN {X 0,Y 455.446,Z 1061.093,A -85,B 0,C 180,E1 21619.56,E2 21619.56} C_VEL
LIN {X 0,Y 454.58,Z 1076.52,A -85,B 0,C 180,E1 21618.599,E2 21618.599} C_VEL
LIN {X 0,Y 453.552,Z 1091.827,A -85,B 0,C 180,E1 21617.38,E2 21617.38} C_VEL
LIN {X 0,Y 452.517,Z 1106.079,A -85,B 0,C 180,E1 21615.968,E2 21615.968} C_VEL
LIN {X 0,Y 451.579,Z 1118.256,A -85,B 0,C 180,E1 21614.489,E2 21614.489} C_VEL
LIN {X 0,Y 450.709,Z 1129.542,A -85,B 0,C 180,E1 21612.817,E2 21612.817} C_VEL
LIN {X 0,Y 449.957,Z 1139.422,A -85,B 0,C 180,E1 21611.017,E2 21611.017} C_VEL
LIN {X 0,Y 449.336,Z 1148.457,A -85,B 0,C 180,E1 21608.961,E2 21608.961} C_VEL
LIN {X 0,Y 448.959,Z 1155.479,A -85,B 0,C 180,E1 21606.907,E2 21606.907} C_VEL
LIN {X 0,Y 448.706,Z 1160.988,A -85,B 0,C 180,E1 21604.73,E2 21604.73} C_VEL
LIN {X 0,Y 448.582,Z 1164.698,A -85,B 0,C 180,E1 21602.555,E2 21602.555} C_VEL
LIN {X 0,Y 448.561,Z 1166.845,A -85,B 0,C 180,E1 21600.256,E2 21600.256} C_VEL
LIN {X 0,Y 448.58,Z 1167.245,A -85,B 0,C 180,E1 21598.084,E2 21598.084} C_VEL
LIN {X 0,Y 448.682,Z 1166.004,A -85,B 0,C 180,E1 21595.911,E2 21595.911} C_VEL
LIN {X 0,Y 448.862,Z 1162.915,A -85,B 0,C 180,E1 21593.606,E2 21593.606} C_VEL
LIN {X 0,Y 449.187,Z 1158.248,A -85,B 0,C 180,E1 21591.423,E2 21591.423} C_VEL
LIN {X 0,Y 449.634,Z 1152.074,A -85,B 0,C 180,E1 21589.364,E2 21589.364} C_VEL
LIN {X 0,Y 450.293,Z 1143.923,A -85,B 0,C 180,E1 21587.302,E2 21587.302} C_VEL
LIN {X 0,Y 451.178,Z 1134.216,A -85,B 0,C 180,E1 21585.367,E2 21585.367} C_VEL
LIN {X 0,Y 452.101,Z 1123.737,A -85,B 0,C 180,E1 21583.688,E2 21583.688} C_VEL
LIN {X 0,Y 453.099,Z 1111.814,A -85,B 0,C 180,E1 21582.138,E2 21582.138} C_VEL
LIN {X 0,Y 454.163,Z 1098.351,A -85,B 0,C 180,E1 21580.717,E2 21580.717} C_VEL
LIN {X 0,Y 455.158,Z 1083.796,A -85,B 0,C 180,E1 21579.49,E2 21579.49} C_VEL
LIN {X 0,Y 455.929,Z 1069.088,A -85,B 0,C 180,E1 21578.517,E2 21578.517} C_VEL
LIN {X 0,Y 456.562,Z 1052.845,A -85,B 0,C 180,E1 21577.703,E2 21577.703} C_VEL
LIN {X 0,Y 456.94,Z 1036.131,A -85,B 0,C 180,E1 21577.114,E2 21577.114} C_VEL
LIN {X 0,Y 458.22,Z 986.997,A -85,B 0,C 180,E1 21576.012,E2 21576.012} C_VEL
LIN {X 0,Y 462.137,Z 908.568,A -85,B 0,C 180,E1 21574.133,E2 21574.133} C_VEL
LIN {X 0,Y 463.891,Z 881.179,A -85,B 0,C 180,E1 21573.442,E2 21573.442} C_VEL
LIN {X 0,Y 468.828,Z 869.095,A -85,B 0,C 180,E1 21572.571,E2 21572.571} C_VEL
LIN {X 0,Y 475.052,Z 841.757,A -85,B 0,C 180,E1 21569.38,E2 21569.38} C_VEL
LIN {X 0,Y 481.464,Z 822.013,A -85,B 0,C 180,E1 21566.895,E2 21566.895} C_VEL
LIN {X 0,Y 488.774,Z 806.037,A -85,B 0,C 180,E1 21564.708,E2 21564.708} C_VEL
LIN {X 0,Y 490.748,Z 802.577,A -85,B 0,C 180,E1 21564.184,E2 21564.184} C_VEL
LIN {X 0,Y 484.55,Z 812.212,A -85,B 0,C 180,E1 21562.798,E2 21562.798} C_VEL
LIN {X 0,Y 480.821,Z 821.473,A -85,B 0,C 180,E1 21561.434,E2 21561.434} C_VEL
LIN {X 0,Y 479.255,Z 831.186,A -85,B 0,C 180,E1 21560.016,E2 21560.016} C_VEL
LIN {X 0,Y 480.016,Z 841.288,A -85,B 0,C 180,E1 21558.579,E2 21558.579} C_VEL
LIN {X 0,Y 482.891,Z 851.142,A -85,B 0,C 180,E1 21557.223,E2 21557.223} C_VEL
LIN {X 0,Y 488.08,Z 861.36,A -85,B 0,C 180,E1 21555.853,E2 21555.853} C_VEL
LIN {X 0,Y 495.334,Z 871.187,A -85,B 0,C 180,E1 21554.558,E2 21554.558} C_VEL
LIN {X 0,Y 504.569,Z 880.527,A -85,B 0,C 180,E1 21553.344,E2 21553.344} C_VEL
LIN {X 0,Y 515.729,Z 889.196,A -85,B 0,C 180,E1 21552.218,E2 21552.218} C_VEL
LIN {X 0,Y 527.866,Z 896.632,A -85,B 0,C 180,E1 21551.255,E2 21551.255} C_VEL
LIN {X 0,Y 506.599,Z 928.765,A -85,B 0,C 180,E1 21550.418,E2 21550.418} C_VEL
LIN {X 0,Y 495.788,Z 948.026,A -85,B 0,C 180,E1 21549.815,E2 21549.815} C_VEL
LIN {X 0,Y 489.059,Z 963.022,A -85,B 0,C 180,E1 21549.254,E2 21549.254} C_VEL
LIN {X 0,Y 486.547,Z 968.772,A -85,B 0,C 180,E1 21549.033,E2 21549.033} C_VEL
LIN {X 0,Y 479.261,Z 984.437,A -85,B 0,C 180,E1 21548.441,E2 21548.441} C_VEL
LIN {X 0,Y 469.984,Z 1011.362,A -85,B 0,C 180,E1 21547.243,E2 21547.243} C_VEL
LIN {X 0,Y 468.266,Z 1026.958,A -85,B 0,C 180,E1 21547.069,E2 21547.069} C_VEL
LIN {X 0,Y 467.512,Z 1059.333,A -85,B 0,C 180,E1 21546.478,E2 21546.478} C_VEL
LIN {X 0,Y 466.318,Z 1083.569,A -85,B 0,C 180,E1 21545.822,E2 21545.822} C_VEL
LIN {X 0,Y 464.892,Z 1107.413,A -85,B 0,C 180,E1 21544.944,E2 21544.944} C_VEL
LIN {X 0,Y 463.3,Z 1130.966,A -85,B 0,C 180,E1 21543.835,E2 21543.835} C_VEL
LIN {X 0,Y 461.561,Z 1153.146,A -85,B 0,C 180,E1 21542.544,E2 21542.544} C_VEL
LIN {X 0,Y 459.751,Z 1174.593,A -85,B 0,C 180,E1 21541.026,E2 21541.026} C_VEL
LIN {X 0,Y 457.937,Z 1194.289,A -85,B 0,C 180,E1 21539.371,E2 21539.371} C_VEL
LIN {X 0,Y 456.07,Z 1213.248,A -85,B 0,C 180,E1 21537.484,E2 21537.484} C_VEL
LIN {X 0,Y 454.403,Z 1229.679,A -85,B 0,C 180,E1 21535.549,E2 21535.549} C_VEL
LIN {X 0,Y 453.101,Z 1242.483,A -85,B 0,C 180,E1 21533.818,E2 21533.818} C_VEL
LIN {X 0,Y 451.873,Z 1254.551,A -85,B 0,C 180,E1 21531.96,E2 21531.96} C_VEL
LIN {X 0,Y 450.981,Z 1263.686,A -85,B 0,C 180,E1 21530.312,E2 21530.312} C_VEL
LIN {X 0,Y 450.069,Z 1272.489,A -85,B 0,C 180,E1 21528.389,E2 21528.389} C_VEL
LIN {X 0,Y 449.101,Z 1283.153,A -85,B 0,C 180,E1 21525.628,E2 21525.628} C_VEL
LIN {X 0,Y 448.532,Z 1290.976,A -85,B 0,C 180,E1 21523.143,E2 21523.143} C_VEL
LIN {X 0,Y 448.202,Z 1297.046,A -85,B 0,C 180,E1 21520.801,E2 21520.801} C_VEL
LIN {X 0,Y 448.014,Z 1302.609,A -85,B 0,C 180,E1 21518.083,E2 21518.083} C_VEL
LIN {X 0,Y 447.93,Z 1306.381,A -85,B 0,C 180,E1 21515.38,E2 21515.38} C_VEL
LIN {X 0,Y 447.904,Z 1308.504,A -85,B 0,C 180,E1 21512.944,E2 21512.944} C_VEL
LIN {X 0,Y 447.896,Z 1309.408,A -85,B 0,C 180,E1 21510.512,E2 21510.512} C_VEL
LIN {X 0,Y 447.904,Z 1308.835,A -85,B 0,C 180,E1 21507.57,E2 21507.57} C_VEL
LIN {X 0,Y 447.918,Z 1306.792,A -85,B 0,C 180,E1 21505.006,E2 21505.006} C_VEL
LIN {X 0,Y 447.972,Z 1303.783,A -85,B 0,C 180,E1 21502.692,E2 21502.692} C_VEL
LIN {X 0,Y 448.127,Z 1299.109,A -85,B 0,C 180,E1 21500.108,E2 21500.108} C_VEL
LIN {X 0,Y 448.473,Z 1292.099,A -85,B 0,C 180,E1 21497.249,E2 21497.249} C_VEL
LIN {X 0,Y 448.967,Z 1284.894,A -85,B 0,C 180,E1 21494.897,E2 21494.897} C_VEL
LIN {X 0,Y 449.711,Z 1276.223,A -85,B 0,C 180,E1 21492.517,E2 21492.517} C_VEL
LIN {X 0,Y 450.878,Z 1264.76,A -85,B 0,C 180,E1 21489.897,E2 21489.897} C_VEL
LIN {X 0,Y 451.963,Z 1253.908,A -85,B 0,C 180,E1 21487.909,E2 21487.909} C_VEL
LIN {X 0,Y 453.289,Z 1241.606,A -85,B 0,C 180,E1 21485.95,E2 21485.95} C_VEL
LIN {X 0,Y 454.974,Z 1226.607,A -85,B 0,C 180,E1 21483.857,E2 21483.857} C_VEL
LIN {X 0,Y 456.998,Z 1208.629,A -85,B 0,C 180,E1 21481.728,E2 21481.728} C_VEL
LIN {X 0,Y 459.008,Z 1191.102,A -85,B 0,C 180,E1 21479.934,E2 21479.934} C_VEL
LIN {X 0,Y 461.234,Z 1170.883,A -85,B 0,C 180,E1 21478.186,E2 21478.186} C_VEL
LIN {X 0,Y 463.492,Z 1149.44,A -85,B 0,C 180,E1 21476.627,E2 21476.627} C_VEL
LIN {X 0,Y 465.622,Z 1127.467,A -85,B 0,C 180,E1 21475.317,E2 21475.317} C_VEL
LIN {X 0,Y 467.588,Z 1105.079,A -85,B 0,C 180,E1 21474.247,E2 21474.247} C_VEL
LIN {X 0,Y 469.231,Z 1082.546,A -85,B 0,C 180,E1 21473.42,E2 21473.42} C_VEL
LIN {X 0,Y 470.65,Z 1058.247,A -85,B 0,C 180,E1 21472.784,E2 21472.784} C_VEL
LIN {X 0,Y 471.937,Z 1021.198,A -85,B 0,C 180,E1 21472.136,E2 21472.136} C_VEL
LIN {X 0,Y 472.439,Z 1018.077,A -85,B 0,C 180,E1 21472.063,E2 21472.063} C_VEL
LIN {X 0,Y 477.303,Z 1003.436,A -85,B 0,C 180,E1 21471.374,E2 21471.374} C_VEL
LIN {X 0,Y 484.214,Z 985.101,A -85,B 0,C 180,E1 21470.584,E2 21470.584} C_VEL
LIN {X 0,Y 492.192,Z 968.136,A -85,B 0,C 180,E1 21469.989,E2 21469.989} C_VEL
LIN {X 0,Y 498.959,Z 952.526,A -85,B 0,C 180,E1 21469.44,E2 21469.44} C_VEL
LIN {X 0,Y 509.328,Z 933.039,A -85,B 0,C 180,E1 21468.923,E2 21468.923} C_VEL
LIN {X 0,Y 529.158,Z 900.712,A -85,B 0,C 180,E1 21468.31,E2 21468.31} C_VEL
LIN {X 0,Y 530.193,Z 898.846,A -85,B 0,C 180,E1 21468.267,E2 21468.267} C_VEL
LIN {X 0,Y 518.857,Z 892.497,A -85,B 0,C 180,E1 21466.915,E2 21466.915} C_VEL
LIN {X 0,Y 508.436,Z 884.175,A -85,B 0,C 180,E1 21465.388,E2 21465.388} C_VEL
LIN {X 0,Y 500.266,Z 874.893,A -85,B 0,C 180,E1 21463.91,E2 21463.91} C_VEL
LIN {X 0,Y 494.078,Z 865.112,A -85,B 0,C 180,E1 21462.525,E2 21462.525} C_VEL
LIN {X 0,Y 488.755,Z 852.893,A -85,B 0,C 180,E1 21460.987,E2 21460.987} C_VEL
LIN {X 0,Y 485.047,Z 838.906,A -85,B 0,C 180,E1 21459.412,E2 21459.412} C_VEL
LIN {X 0,Y 483.041,Z 823.357,A -85,B 0,C 180,E1 21457.86,E2 21457.86} C_VEL
LIN {X 0,Y 482.787,Z 806.27,A -85,B 0,C 180,E1 21456.331,E2 21456.331} C_VEL
LIN {X 0,Y 484.579,Z 783.444,A -85,B 0,C 180,E1 21454.506,E2 21454.506} C_VEL
LIN {X 0,Y 488.104,Z 749.576,A -85,B 0,C 180,E1 21451.835,E2 21451.835} C_VEL
LIN {X 0,Y 478.345,Z 731.224,A -85,B 0,C 180,E1 21448.598,E2 21448.598} C_VEL
LIN {X 0,Y 470.444,Z 716.891,A -85,B 0,C 180,E1 21445.829,E2 21445.829} C_VEL
LIN {X 0,Y 463.209,Z 703.852,A -85,B 0,C 180,E1 21443.132,E2 21443.132} C_VEL
LIN {X 0,Y 459.448,Z 697.568,A -85,B 0,C 180,E1 21441.713,E2 21441.713} C_VEL
LIN {X 0,Y 457.043,Z 693.304,A -85,B 0,C 180,E1 21440.757,E2 21440.757} C_VEL
LIN {X 0,Y 454.433,Z 688.616,A -85,B 0,C 180,E1 21439.672,E2 21439.672} C_VEL
LIN {X 0,Y 452.339,Z 685.125,A -85,B 0,C 180,E1 21438.827,E2 21438.827} C_VEL
LIN {X 0,Y 451.507,Z 683.553,A -85,B 0,C 180,E1 21438.462,E2 21438.462} C_VEL
LIN {X 0,Y 449.446,Z 680.227,A -85,B 0,C 180,E1 21437.611,E2 21437.611} C_VEL
LIN {X 0,Y 449.123,Z 678.788,A -85,B 0,C 180,E1 21437.323,E2 21437.323} C_VEL
LIN {X 0,Y 449.13,Z 678.788,A -85,B 0,C 180,E1 21433.649,E2 21433.649} C_VEL
LIN {X 0,Y 449.128,Z 678.788,A -85,B 0,C 180,E1 21430,E2 21430} C_VEL
LIN {X 0,Y 449.125,Z 678.786,A -85,B 0,C 180,E1 21426.262,E2 21426.262} C_VEL
LIN {X 0,Y 449.128,Z 678.787,A -85,B 0,C 180,E1 21422.552,E2 21422.552} C_VEL
LIN {X 0,Y 449.123,Z 678.79,A -85,B 0,C 180,E1 21418.852,E2 21418.852} C_VEL
LIN {X 0,Y 449.137,Z 678.791,A -85,B 0,C 180,E1 21415.019,E2 21415.019} C_VEL
LIN {X 0,Y 449.123,Z 678.788,A -85,B 0,C 180,E1 21411.279,E2 21411.279} C_VEL
LIN {X 0,Y 449.139,Z 678.791,A -85,B 0,C 180,E1 21407.529,E2 21407.529} C_VEL
LIN {X 0,Y 449.133,Z 678.789,A -85,B 0,C 180,E1 21403.842,E2 21403.842} C_VEL
LIN {X 0,Y 449.132,Z 678.781,A -85,B 0,C 180,E1 21400.086,E2 21400.086} C_VEL
LIN {X 0,Y 449.132,Z 678.78,A -85,B 0,C 180,E1 21396.377,E2 21396.377} C_VEL
LIN {X 0,Y 449.135,Z 678.758,A -85,B 0,C 180,E1 21392.56,E2 21392.56} C_VEL
LIN {X 0,Y 449.14,Z 678.781,A -85,B 0,C 180,E1 21388.741,E2 21388.741} C_VEL
LIN {X 0,Y 449.126,Z 678.751,A -85,B 0,C 180,E1 21384.944,E2 21384.944} C_VEL
LIN {X 0,Y 449.14,Z 678.784,A -85,B 0,C 180,E1 21381.113,E2 21381.113} C_VEL
LIN {X 0,Y 449.131,Z 678.786,A -85,B 0,C 180,E1 21377.235,E2 21377.235} C_VEL
LIN {X 0,Y 449.144,Z 678.911,A -85,B 0,C 180,E1 21376.755,E2 21376.755} C_VEL
LIN {X 0,Y 450.356,Z 682.148,A -85,B 0,C 180,E1 21376.333,E2 21376.333} C_VEL
LIN {X 0,Y 451.518,Z 684.076,A -85,B 0,C 180,E1 21376.028,E2 21376.028} C_VEL
LIN {X 0,Y 459.302,Z 700.156,A -85,B 0,C 180,E1 21373.719,E2 21373.719} C_VEL
LIN {X 0,Y 467.016,Z 717.819,A -85,B 0,C 180,E1 21371.384,E2 21371.384} C_VEL
LIN {X 0,Y 470.759,Z 727.143,A -85,B 0,C 180,E1 21370.215,E2 21370.215} C_VEL
LIN {X 0,Y 468.77,Z 767.366,A -85,B 0,C 180,E1 21367.282,E2 21367.282} C_VEL
LIN {X 0,Y 468.782,Z 772.302,A -85,B 0,C 180,E1 21366.977,E2 21366.977} C_VEL
LIN {X 0,Y 471.614,Z 792.28,A -85,B 0,C 180,E1 21366.341,E2 21366.341} C_VEL
LIN {X 0,Y 469.775,Z 878.313,A -85,B 0,C 180,E1 21364.909,E2 21364.909} C_VEL
LIN {X 0,Y 468.797,Z 886.004,A -85,B 0,C 180,E1 21364.852,E2 21364.852} C_VEL
LIN {X 0,Y 463.264,Z 906.502,A -85,B 0,C 180,E1 21364.954,E2 21364.954} C_VEL
LIN {X 0,Y 462.51,Z 913.102,A -85,B 0,C 180,E1 21364.897,E2 21364.897} C_VEL
LIN {X 0,Y 459.865,Z 1033.749,A -85,B 0,C 180,E1 21362.847,E2 21362.847} C_VEL
LIN {X 0,Y 458.928,Z 1054.326,A -85,B 0,C 180,E1 21362.281,E2 21362.281} C_VEL
LIN {X 0,Y 457.623,Z 1074.734,A -85,B 0,C 180,E1 21361.478,E2 21361.478} C_VEL
LIN {X 0,Y 456.03,Z 1093.809,A -85,B 0,C 180,E1 21360.496,E2 21360.496} C_VEL
LIN {X 0,Y 454.254,Z 1111.986,A -85,B 0,C 180,E1 21359.323,E2 21359.323} C_VEL
LIN {X 0,Y 452.215,Z 1130.173,A -85,B 0,C 180,E1 21357.88,E2 21357.88} C_VEL
LIN {X 0,Y 450.105,Z 1147.257,A -85,B 0,C 180,E1 21356.234,E2 21356.234} C_VEL
LIN {X 0,Y 448.05,Z 1162.949,A -85,B 0,C 180,E1 21354.427,E2 21354.427} C_VEL
LIN {X 0,Y 446.223,Z 1176.868,A -85,B 0,C 180,E1 21352.529,E2 21352.529} C_VEL
LIN {X 0,Y 444.52,Z 1190.068,A -85,B 0,C 180,E1 21350.404,E2 21350.404} C_VEL
LIN {X 0,Y 443.08,Z 1201.874,A -85,B 0,C 180,E1 21348.144,E2 21348.144} C_VEL
LIN {X 0,Y 441.932,Z 1212.276,A -85,B 0,C 180,E1 21345.753,E2 21345.753} C_VEL
LIN {X 0,Y 441.042,Z 1221.63,A -85,B 0,C 180,E1 21343.102,E2 21343.102} C_VEL
LIN {X 0,Y 440.502,Z 1228.636,A -85,B 0,C 180,E1 21340.594,E2 21340.594} C_VEL
LIN {X 0,Y 440.197,Z 1234.274,A -85,B 0,C 180,E1 21337.964,E2 21337.964} C_VEL
LIN {X 0,Y 440.037,Z 1238.404,A -85,B 0,C 180,E1 21335.214,E2 21335.214} C_VEL
LIN {X 0,Y 439.992,Z 1240.738,A -85,B 0,C 180,E1 21332.604,E2 21332.604} C_VEL
LIN {X 0,Y 439.987,Z 1241.556,A -85,B 0,C 180,E1 21329.999,E2 21329.999} C_VEL
LIN {X 0,Y 439.992,Z 1240.719,A -85,B 0,C 180,E1 21327.264,E2 21327.264} C_VEL
LIN {X 0,Y 440.04,Z 1238.358,A -85,B 0,C 180,E1 21324.654,E2 21324.654} C_VEL
LIN {X 0,Y 440.199,Z 1234.194,A -85,B 0,C 180,E1 21321.904,E2 21321.904} C_VEL
LIN {X 0,Y 440.507,Z 1228.521,A -85,B 0,C 180,E1 21319.273,E2 21319.273} C_VEL
LIN {X 0,Y 441.056,Z 1221.482,A -85,B 0,C 180,E1 21316.763,E2 21316.763} C_VEL
LIN {X 0,Y 441.896,Z 1212.618,A -85,B 0,C 180,E1 21314.245,E2 21314.245} C_VEL
LIN {X 0,Y 443.045,Z 1202.147,A -85,B 0,C 180,E1 21311.825,E2 21311.825} C_VEL
LIN {X 0,Y 444.453,Z 1190.548,A -85,B 0,C 180,E1 21309.592,E2 21309.592} C_VEL
LIN {X 0,Y 446.206,Z 1177.005,A -85,B 0,C 180,E1 21307.401,E2 21307.401} C_VEL
LIN {X 0,Y 448.198,Z 1161.827,A -85,B 0,C 180,E1 21305.344,E2 21305.344} C_VEL
LIN {X 0,Y 450.241,Z 1146.136,A -85,B 0,C 180,E1 21303.56,E2 21303.56} C_VEL
LIN {X 0,Y 452.281,Z 1129.589,A -85,B 0,C 180,E1 21301.98,E2 21301.98} C_VEL
LIN {X 0,Y 454.335,Z 1111.318,A -85,B 0,C 180,E1 21300.537,E2 21300.537} C_VEL
LIN {X 0,Y 456.242,Z 1091.811,A -85,B 0,C 180,E1 21299.294,E2 21299.294} C_VEL
LIN {X 0,Y 457.816,Z 1072.215,A -85,B 0,C 180,E1 21298.315,E2 21298.315} C_VEL
LIN {X 0,Y 459.048,Z 1052.344,A -85,B 0,C 180,E1 21297.563,E2 21297.563} C_VEL
LIN {X 0,Y 459.935,Z 1031.523,A -85,B 0,C 180,E1 21297.015,E2 21297.015} C_VEL
LIN {X 0,Y 465.039,Z 800.395,A -85,B 0,C 180,E1 21293.113,E2 21293.113} C_VEL
LIN {X 0,Y 459.037,Z 773.628,A -85,B 0,C 180,E1 21291.988,E2 21291.988} C_VEL
LIN {X 0,Y 460.405,Z 745.596,A -85,B 0,C 180,E1 21289.091,E2 21289.091} C_VEL
LIN {X 0,Y 461.356,Z 730.672,A -85,B 0,C 180,E1 21287.454,E2 21287.454} C_VEL
LIN {X 0,Y 454.673,Z 711.594,A -85,B 0,C 180,E1 21284.372,E2 21284.372} C_VEL
LIN {X 0,Y 448.943,Z 697.513,A -85,B 0,C 180,E1 21281.926,E2 21281.926} C_VEL
LIN {X 0,Y 455.818,Z 713.757,A -85,B 0,C 180,E1 21279.256,E2 21279.256} C_VEL
LIN {X 0,Y 461.886,Z 729.644,A -85,B 0,C 180,E1 21276.844,E2 21276.844} C_VEL
LIN {X 0,Y 458.605,Z 768,A -85,B 0,C 180,E1 21273.111,E2 21273.111} C_VEL
LIN {X 0,Y 455.346,Z 809.131,A -85,B 0,C 180,E1 21269.175,E2 21269.175} C_VEL
LIN {X 0,Y 452.41,Z 849.955,A -85,B 0,C 180,E1 21265.321,E2 21265.321} C_VEL
LIN {X 0,Y 452.086,Z 856.857,A -85,B 0,C 180,E1 21264.709,E2 21264.709} C_VEL
LIN {X 0,Y 453.331,Z 866.437,A -85,B 0,C 180,E1 21264.422,E2 21264.422} C_VEL
LIN {X 0,Y 449.276,Z 1027.547,A -85,B 0,C 180,E1 21261.3,E2 21261.3} C_VEL
LIN {X 0,Y 448.733,Z 1045.579,A -85,B 0,C 180,E1 21260.694,E2 21260.694} C_VEL
LIN {X 0,Y 447.979,Z 1062.149,A -85,B 0,C 180,E1 21259.9,E2 21259.9} C_VEL
LIN {X 0,Y 447.055,Z 1077.84,A -85,B 0,C 180,E1 21258.904,E2 21258.904} C_VEL
LIN {X 0,Y 445.979,Z 1093.084,A -85,B 0,C 180,E1 21257.668,E2 21257.668} C_VEL
LIN {X 0,Y 444.855,Z 1107.766,A -85,B 0,C 180,E1 21256.183,E2 21256.183} C_VEL
LIN {X 0,Y 443.835,Z 1120.351,A -85,B 0,C 180,E1 21254.615,E2 21254.615} C_VEL
LIN {X 0,Y 442.922,Z 1131.458,A -85,B 0,C 180,E1 21252.914,E2 21252.914} C_VEL
LIN {X 0,Y 442.089,Z 1141.865,A -85,B 0,C 180,E1 21250.952,E2 21250.952} C_VEL
LIN {X 0,Y 441.465,Z 1150.705,A -85,B 0,C 180,E1 21248.86,E2 21248.86} C_VEL
LIN {X 0,Y 441.075,Z 1157.496,A -85,B 0,C 180,E1 21246.77,E2 21246.77} C_VEL
LIN {X 0,Y 440.808,Z 1162.806,A -85,B 0,C 180,E1 21244.554,E2 21244.554} C_VEL
LIN {X 0,Y 440.7,Z 1166.368,A -85,B 0,C 180,E1 21242.341,E2 21242.341} C_VEL
LIN {X 0,Y 440.679,Z 1168.299,A -85,B 0,C 180,E1 21240.13,E2 21240.13} C_VEL
LIN {X 0,Y 440.711,Z 1168.609,A -85,B 0,C 180,E1 21237.92,E2 21237.92} C_VEL
LIN {X 0,Y 440.834,Z 1167.155,A -85,B 0,C 180,E1 21235.578,E2 21235.578} C_VEL
LIN {X 0,Y 441.048,Z 1164.141,A -85,B 0,C 180,E1 21233.361,E2 21233.361} C_VEL
LIN {X 0,Y 441.422,Z 1159.375,A -85,B 0,C 180,E1 21231.14,E2 21231.14} C_VEL
LIN {X 0,Y 441.956,Z 1152.62,A -85,B 0,C 180,E1 21228.913,E2 21228.913} C_VEL
LIN {X 0,Y 442.744,Z 1144.291,A -85,B 0,C 180,E1 21226.816,E2 21226.816} C_VEL
LIN {X 0,Y 443.652,Z 1135.016,A -85,B 0,C 180,E1 21224.979,E2 21224.979} C_VEL
LIN {X 0,Y 444.643,Z 1124.345,A -85,B 0,C 180,E1 21223.272,E2 21223.272} C_VEL
LIN {X 0,Y 445.788,Z 1111.736,A -85,B 0,C 180,E1 21221.632,E2 21221.632} C_VEL
LIN {X 0,Y 446.888,Z 1098.634,A -85,B 0,C 180,E1 21220.255,E2 21220.255} C_VEL
LIN {X 0,Y 447.873,Z 1084.517,A -85,B 0,C 180,E1 21219.072,E2 21219.072} C_VEL
LIN {X 0,Y 448.747,Z 1068.499,A -85,B 0,C 180,E1 21218.018,E2 21218.018} C_VEL
LIN {X 0,Y 449.377,Z 1052.421,A -85,B 0,C 180,E1 21217.227,E2 21217.227} C_VEL
LIN {X 0,Y 449.704,Z 1035.537,A -85,B 0,C 180,E1 21216.66,E2 21216.66} C_VEL
LIN {X 0,Y 451.313,Z 986.02,A -85,B 0,C 180,E1 21215.487,E2 21215.487} C_VEL
LIN {X 0,Y 455.859,Z 908.322,A -85,B 0,C 180,E1 21213.506,E2 21213.506} C_VEL
LIN {X 0,Y 457.53,Z 885.141,A -85,B 0,C 180,E1 21212.894,E2 21212.894} C_VEL
LIN {X 0,Y 463.396,Z 871.226,A -85,B 0,C 180,E1 21211.872,E2 21211.872} C_VEL
LIN {X 0,Y 469.959,Z 845.558,A -85,B 0,C 180,E1 21208.79,E2 21208.79} C_VEL
LIN {X 0,Y 476.785,Z 826.848,A -85,B 0,C 180,E1 21206.361,E2 21206.361} C_VEL
LIN {X 0,Y 484.409,Z 811.928,A -85,B 0,C 180,E1 21204.258,E2 21204.258} C_VEL
LIN {X 0,Y 484.453,Z 811.83,A -85,B 0,C 180,E1 21204.205,E2 21204.205} C_VEL
LIN {X 0,Y 478.511,Z 821.312,A -85,B 0,C 180,E1 21202.76,E2 21202.76} C_VEL
LIN {X 0,Y 475.081,Z 830.598,A -85,B 0,C 180,E1 21201.313,E2 21201.313} C_VEL
LIN {X 0,Y 473.966,Z 839.438,A -85,B 0,C 180,E1 21199.953,E2 21199.953} C_VEL
LIN {X 0,Y 475.032,Z 849.369,A -85,B 0,C 180,E1 21198.47,E2 21198.47} C_VEL
LIN {X 0,Y 478.339,Z 859.249,A -85,B 0,C 180,E1 21197.045,E2 21197.045} C_VEL
LIN {X 0,Y 483.726,Z 868.991,A -85,B 0,C 180,E1 21195.682,E2 21195.682} C_VEL
LIN {X 0,Y 491.721,Z 879.148,A -85,B 0,C 180,E1 21194.296,E2 21194.296} C_VEL
LIN {X 0,Y 501.123,Z 888.101,A -85,B 0,C 180,E1 21193.092,E2 21193.092} C_VEL
LIN {X 0,Y 512.386,Z 896.481,A -85,B 0,C 180,E1 21191.972,E2 21191.972} C_VEL
LIN {X 0,Y 517.404,Z 899.778,A -85,B 0,C 180,E1 21191.544,E2 21191.544} C_VEL
LIN {X 0,Y 499.276,Z 927.666,A -85,B 0,C 180,E1 21190.833,E2 21190.833} C_VEL
LIN {X 0,Y 488.942,Z 946.291,A -85,B 0,C 180,E1 21190.256,E2 21190.256} C_VEL
LIN {X 0,Y 481.839,Z 962.242,A -85,B 0,C 180,E1 21189.659,E2 21189.659} C_VEL
LIN {X 0,Y 477.811,Z 970.69,A -85,B 0,C 180,E1 21189.35,E2 21189.35} C_VEL
LIN {X 0,Y 470.783,Z 986.836,A -85,B 0,C 180,E1 21188.717,E2 21188.717} C_VEL
LIN {X 0,Y 463.131,Z 1009.513,A -85,B 0,C 180,E1 21187.724,E2 21187.724} C_VEL
LIN {X 0,Y 461.173,Z 1026.837,A -85,B 0,C 180,E1 21187.528,E2 21187.528} C_VEL
LIN {X 0,Y 460.335,Z 1057.98,A -85,B 0,C 180,E1 21186.932,E2 21186.932} C_VEL
LIN {X 0,Y 458.95,Z 1083.151,A -85,B 0,C 180,E1 21186.219,E2 21186.219} C_VEL
LIN {X 0,Y 457.323,Z 1108.338,A -85,B 0,C 180,E1 21185.254,E2 21185.254} C_VEL
LIN {X 0,Y 455.664,Z 1131.226,A -85,B 0,C 180,E1 21184.132,E2 21184.132} C_VEL
LIN {X 0,Y 453.848,Z 1153.063,A -85,B 0,C 180,E1 21182.817,E2 21182.817} C_VEL
LIN {X 0,Y 451.951,Z 1174.672,A -85,B 0,C 180,E1 21181.251,E2 21181.251} C_VEL
LIN {X 0,Y 450.065,Z 1194.445,A -85,B 0,C 180,E1 21179.551,E2 21179.551} C_VEL
LIN {X 0,Y 448.048,Z 1214.323,A -85,B 0,C 180,E1 21177.513,E2 21177.513} C_VEL
LIN {X 0,Y 446.411,Z 1229.972,A -85,B 0,C 180,E1 21175.613,E2 21175.613} C_VEL
LIN {X 0,Y 445.093,Z 1242.672,A -85,B 0,C 180,E1 21173.851,E2 21173.851} C_VEL
LIN {X 0,Y 443.707,Z 1256.295,A -85,B 0,C 180,E1 21171.689,E2 21171.689} C_VEL
LIN {X 0,Y 442.515,Z 1268.411,A -85,B 0,C 180,E1 21169.4,E2 21169.4} C_VEL
LIN {X 0,Y 441.739,Z 1276.979,A -85,B 0,C 180,E1 21167.521,E2 21167.521} C_VEL
LIN {X 0,Y 441.136,Z 1284.016,A -85,B 0,C 180,E1 21165.648,E2 21165.648} C_VEL
LIN {X 0,Y 440.595,Z 1290.971,A -85,B 0,C 180,E1 21163.384,E2 21163.384} C_VEL
LIN {X 0,Y 440.25,Z 1296.734,A -85,B 0,C 180,E1 21161.131,E2 21161.131} C_VEL
LIN {X 0,Y 440.034,Z 1301.873,A -85,B 0,C 180,E1 21158.626,E2 21158.626} C_VEL
LIN {X 0,Y 439.935,Z 1306.103,A -85,B 0,C 180,E1 21155.74,E2 21155.74} C_VEL
LIN {X 0,Y 439.911,Z 1308.337,A -85,B 0,C 180,E1 21153.258,E2 21153.258} C_VEL
LIN {X 0,Y 439.904,Z 1309.324,A -85,B 0,C 180,E1 21150.912,E2 21150.912} C_VEL
LIN {X 0,Y 439.901,Z 1309.212,A -85,B 0,C 180,E1 21148.568,E2 21148.568} C_VEL
LIN {X 0,Y 439.913,Z 1307.617,A -85,B 0,C 180,E1 21145.699,E2 21145.699} C_VEL
LIN {X 0,Y 439.97,Z 1304.364,A -85,B 0,C 180,E1 21142.952,E2 21142.952} C_VEL
LIN {X 0,Y 440.094,Z 1300.37,A -85,B 0,C 180,E1 21140.586,E2 21140.586} C_VEL
LIN {X 0,Y 440.35,Z 1294.998,A -85,B 0,C 180,E1 21138.131,E2 21138.131} C_VEL
LIN {X 0,Y 440.926,Z 1286.639,A -85,B 0,C 180,E1 21135.153,E2 21135.153} C_VEL
LIN {X 0,Y 441.508,Z 1279.685,A -85,B 0,C 180,E1 21133.15,E2 21133.15} C_VEL
LIN {X 0,Y 442.331,Z 1270.516,A -85,B 0,C 180,E1 21131.005,E2 21131.005} C_VEL
LIN {X 0,Y 443.329,Z 1260.576,A -85,B 0,C 180,E1 21128.987,E2 21128.987} C_VEL
LIN {X 0,Y 444.755,Z 1247.626,A -85,B 0,C 180,E1 21126.693,E2 21126.693} C_VEL
LIN {X 0,Y 446.549,Z 1231.848,A -85,B 0,C 180,E1 21124.326,E2 21124.326} C_VEL
LIN {X 0,Y 448.34,Z 1216.723,A -85,B 0,C 180,E1 21122.364,E2 21122.364} C_VEL
LIN {X 0,Y 450.623,Z 1198,A -85,B 0,C 180,E1 21120.273,E2 21120.273} C_VEL
LIN {X 0,Y 452.92,Z 1178.628,A -85,B 0,C 180,E1 21118.443,E2 21118.443} C_VEL
LIN {X 0,Y 455.279,Z 1157.639,A -85,B 0,C 180,E1 21116.775,E2 21116.775} C_VEL
LIN {X 0,Y 457.647,Z 1136.027,A -85,B 0,C 180,E1 21115.348,E2 21115.348} C_VEL
LIN {X 0,Y 459.782,Z 1113.942,A -85,B 0,C 180,E1 21114.161,E2 21114.161} C_VEL
LIN {X 0,Y 461.748,Z 1090.878,A -85,B 0,C 180,E1 21113.198,E2 21113.198} C_VEL
LIN {X 0,Y 463.341,Z 1068.031,A -85,B 0,C 180,E1 21112.491,E2 21112.491} C_VEL
LIN {X 0,Y 464.407,Z 1044.582,A -85,B 0,C 180,E1 21111.985,E2 21111.985} C_VEL
LIN {X 0,Y 465.355,Z 1020.762,A -85,B 0,C 180,E1 21111.582,E2 21111.582} C_VEL
LIN {X 0,Y 465.871,Z 1017.201,A -85,B 0,C 180,E1 21111.509,E2 21111.509} C_VEL
LIN {X 0,Y 470.803,Z 1002.591,A -85,B 0,C 180,E1 21110.819,E2 21110.819} C_VEL
LIN {X 0,Y 477.783,Z 984.222,A -85,B 0,C 180,E1 21110.025,E2 21110.025} C_VEL
LIN {X 0,Y 485.814,Z 967.28,A -85,B 0,C 180,E1 21109.432,E2 21109.432} C_VEL
LIN {X 0,Y 492.567,Z 951.864,A -85,B 0,C 180,E1 21108.877,E2 21108.877} C_VEL
LIN {X 0,Y 502.653,Z 932.771,A -85,B 0,C 180,E1 21108.366,E2 21108.366} C_VEL
LIN {X 0,Y 519.749,Z 904.663,A -85,B 0,C 180,E1 21107.827,E2 21107.827} C_VEL
LIN {X 0,Y 520.666,Z 902.881,A -85,B 0,C 180,E1 21107.78,E2 21107.78} C_VEL
LIN {X 0,Y 509.783,Z 895.816,A -85,B 0,C 180,E1 21106.363,E2 21106.363} C_VEL
LIN {X 0,Y 500.338,Z 887.307,A -85,B 0,C 180,E1 21104.863,E2 21104.863} C_VEL
LIN {X 0,Y 491.987,Z 876.705,A -85,B 0,C 180,E1 21103.226,E2 21103.226} C_VEL
LIN {X 0,Y 485.652,Z 865.049,A -85,B 0,C 180,E1 21101.64,E2 21101.64} C_VEL
LIN {X 0,Y 480.961,Z 851.947,A -85,B 0,C 180,E1 21100.046,E2 21100.046} C_VEL
LIN {X 0,Y 477.861,Z 836.94,A -85,B 0,C 180,E1 21098.42,E2 21098.42} C_VEL
LIN {X 0,Y 476.543,Z 820.209,A -85,B 0,C 180,E1 21096.8,E2 21096.8} C_VEL
LIN {X 0,Y 477.128,Z 800.807,A -85,B 0,C 180,E1 21095.123,E2 21095.123} C_VEL
LIN {X 0,Y 482.128,Z 754.087,A -85,B 0,C 180,E1 21091.42,E2 21091.42} C_VEL
LIN {X 0,Y 472.457,Z 735.848,A -85,B 0,C 180,E1 21088.16,E2 21088.16} C_VEL
LIN {X 0,Y 464.912,Z 722.096,A -85,B 0,C 180,E1 21085.475,E2 21085.475} C_VEL
LIN {X 0,Y 457.998,Z 709.615,A -85,B 0,C 180,E1 21082.867,E2 21082.867} C_VEL
LIN {X 0,Y 452.176,Z 699.505,A -85,B 0,C 180,E1 21080.584,E2 21080.584} C_VEL
LIN {X 0,Y 449.189,Z 694.38,A -85,B 0,C 180,E1 21079.369,E2 21079.369} C_VEL
LIN {X 0,Y 446.627,Z 689.76,A -85,B 0,C 180,E1 21078.265,E2 21078.265} C_VEL
LIN {X 0,Y 444.545,Z 686.414,A -85,B 0,C 180,E1 21077.406,E2 21077.406} C_VEL
LIN {X 0,Y 443.79,Z 684.748,A -85,B 0,C 180,E1 21077.031,E2 21077.031} C_VEL
LIN {X 0,Y 441.665,Z 681.669,A -85,B 0,C 180,E1 21076.168,E2 21076.168} C_VEL
LIN {X 0,Y 441.196,Z 679.776,A -85,B 0,C 180,E1 21075.78,E2 21075.78} C_VEL
LIN {X 0,Y 441.198,Z 679.776,A -85,B 0,C 180,E1 21071.901,E2 21071.901} C_VEL
LIN {X 0,Y 441.196,Z 679.775,A -85,B 0,C 180,E1 21068.077,E2 21068.077} C_VEL
LIN {X 0,Y 441.197,Z 679.775,A -85,B 0,C 180,E1 21064.289,E2 21064.289} C_VEL
LIN {X 0,Y 441.196,Z 679.773,A -85,B 0,C 180,E1 21060.389,E2 21060.389} C_VEL
LIN {X 0,Y 441.192,Z 679.778,A -85,B 0,C 180,E1 21056.622,E2 21056.622} C_VEL
LIN {X 0,Y 441.195,Z 679.779,A -85,B 0,C 180,E1 21052.84,E2 21052.84} C_VEL
LIN {X 0,Y 441.192,Z 679.776,A -85,B 0,C 180,E1 21049.026,E2 21049.026} C_VEL
LIN {X 0,Y 441.194,Z 679.779,A -85,B 0,C 180,E1 21045.296,E2 21045.296} C_VEL
LIN {X 0,Y 441.186,Z 679.771,A -85,B 0,C 180,E1 21041.501,E2 21041.501} C_VEL
LIN {X 0,Y 441.192,Z 679.774,A -85,B 0,C 180,E1 21037.761,E2 21037.761} C_VEL
LIN {X 0,Y 441.186,Z 679.779,A -85,B 0,C 180,E1 21034.062,E2 21034.062} C_VEL
LIN {X 0,Y 441.192,Z 679.732,A -85,B 0,C 180,E1 21030.393,E2 21030.393} C_VEL
LIN {X 0,Y 441.187,Z 679.772,A -85,B 0,C 180,E1 21026.739,E2 21026.739} C_VEL
LIN {X 0,Y 441.194,Z 679.76,A -85,B 0,C 180,E1 21022.912,E2 21022.912} C_VEL
LIN {X 0,Y 441.183,Z 679.743,A -85,B 0,C 180,E1 21019.195,E2 21019.195} C_VEL
LIN {X 0,Y 441.225,Z 679.949,A -85,B 0,C 180,E1 21017.698,E2 21017.698} C_VEL
LIN {X 0,Y 442.477,Z 683.226,A -85,B 0,C 180,E1 21017.255,E2 21017.255} C_VEL
LIN {X 0,Y 443.667,Z 685.15,A -85,B 0,C 180,E1 21016.933,E2 21016.933} C_VEL
LIN {X 0,Y 451.816,Z 701.728,A -85,B 0,C 180,E1 21014.464,E2 21014.464} C_VEL
LIN {X 0,Y 459.611,Z 719.312,A -85,B 0,C 180,E1 21012.069,E2 21012.069} C_VEL
LIN {X 0,Y 464.158,Z 730.462,A -85,B 0,C 180,E1 21010.637,E2 21010.637} C_VEL
LIN {X 0,Y 462.244,Z 768.946,A -85,B 0,C 180,E1 21007.822,E2 21007.822} C_VEL
LIN {X 0,Y 462.291,Z 772.919,A -85,B 0,C 180,E1 21007.583,E2 21007.583} C_VEL
LIN {X 0,Y 465.186,Z 793.581,A -85,B 0,C 180,E1 21006.91,E2 21006.91} C_VEL
LIN {X 0,Y 462.51,Z 913.102,A -85,B 0,C 180,E1 21004.897,E2 21004.897} C_VEL
LIN {X 0,Y 461.523,Z 920.792,A -85,B 0,C 180,E1 21004.84,E2 21004.84} C_VEL
LIN {X 0,Y 455.936,Z 941.279,A -85,B 0,C 180,E1 21004.948,E2 21004.948} C_VEL
LIN {X 0,Y 455.183,Z 947.878,A -85,B 0,C 180,E1 21004.89,E2 21004.89} C_VEL
LIN {X 0,Y 453.165,Z 1034.649,A -85,B 0,C 180,E1 21003.386,E2 21003.386} C_VEL
LIN {X 0,Y 452.18,Z 1055.205,A -85,B 0,C 180,E1 21002.81,E2 21002.81} C_VEL
LIN {X 0,Y 450.827,Z 1075.305,A -85,B 0,C 180,E1 21002.009,E2 21002.009} C_VEL
LIN {X 0,Y 449.156,Z 1094.393,A -85,B 0,C 180,E1 21001.014,E2 21001.014} C_VEL
LIN {X 0,Y 447.282,Z 1112.578,A -85,B 0,C 180,E1 20999.826,E2 20999.826} C_VEL
LIN {X 0,Y 445.174,Z 1130.405,A -85,B 0,C 180,E1 20998.394,E2 20998.394} C_VEL
LIN {X 0,Y 442.96,Z 1147.343,A -85,B 0,C 180,E1 20996.749,E2 20996.749} C_VEL
LIN {X 0,Y 440.821,Z 1162.821,A -85,B 0,C 180,E1 20994.953,E2 20994.953} C_VEL
LIN {X 0,Y 438.774,Z 1177.477,A -85,B 0,C 180,E1 20992.933,E2 20992.933} C_VEL
LIN {X 0,Y 436.948,Z 1190.679,A -85,B 0,C 180,E1 20990.773,E2 20990.773} C_VEL
LIN {X 0,Y 435.4,Z 1202.486,A -85,B 0,C 180,E1 20988.475,E2 20988.475} C_VEL
LIN {X 0,Y 434.154,Z 1212.889,A -85,B 0,C 180,E1 20986.042,E2 20986.042} C_VEL
LIN {X 0,Y 433.188,Z 1222.243,A -85,B 0,C 180,E1 20983.344,E2 20983.344} C_VEL
LIN {X 0,Y 432.594,Z 1229.249,A -85,B 0,C 180,E1 20980.79,E2 20980.79} C_VEL
LIN {X 0,Y 432.247,Z 1234.917,A -85,B 0,C 180,E1 20978.094,E2 20978.094} C_VEL
LIN {X 0,Y 432.071,Z 1239.015,A -85,B 0,C 180,E1 20975.311,E2 20975.311} C_VEL
LIN {X 0,Y 432.018,Z 1241.347,A -85,B 0,C 180,E1 20972.652,E2 20972.652} C_VEL
LIN {X 0,Y 432.011,Z 1242.165,A -85,B 0,C 180,E1 20969.999,E2 20969.999} C_VEL
LIN {X 0,Y 432.018,Z 1241.327,A -85,B 0,C 180,E1 20967.214,E2 20967.214} C_VEL
LIN {X 0,Y 432.074,Z 1238.967,A -85,B 0,C 180,E1 20964.555,E2 20964.555} C_VEL
LIN {X 0,Y 432.251,Z 1234.803,A -85,B 0,C 180,E1 20961.754,E2 20961.754} C_VEL
LIN {X 0,Y 432.6,Z 1229.131,A -85,B 0,C 180,E1 20959.074,E2 20959.074} C_VEL
LIN {X 0,Y 433.201,Z 1222.09,A -85,B 0,C 180,E1 20956.519,E2 20956.519} C_VEL
LIN {X 0,Y 434.118,Z 1213.224,A -85,B 0,C 180,E1 20953.955,E2 20953.955} C_VEL
LIN {X 0,Y 435.429,Z 1202.267,A -85,B 0,C 180,E1 20951.386,E2 20951.386} C_VEL
LIN {X 0,Y 436.982,Z 1190.409,A -85,B 0,C 180,E1 20949.087,E2 20949.087} C_VEL
LIN {X 0,Y 438.822,Z 1177.15,A -85,B 0,C 180,E1 20946.927,E2 20946.927} C_VEL
LIN {X 0,Y 440.88,Z 1162.423,A -85,B 0,C 180,E1 20944.906,E2 20944.906} C_VEL
LIN {X 0,Y 443.049,Z 1146.662,A -85,B 0,C 180,E1 20943.089,E2 20943.089} C_VEL
LIN {X 0,Y 445.205,Z 1130.172,A -85,B 0,C 180,E1 20941.494,E2 20941.494} C_VEL
LIN {X 0,Y 447.37,Z 1111.893,A -85,B 0,C 180,E1 20940.032,E2 20940.032} C_VEL
LIN {X 0,Y 449.264,Z 1093.468,A -85,B 0,C 180,E1 20938.839,E2 20938.839} C_VEL
LIN {X 0,Y 450.869,Z 1074.883,A -85,B 0,C 180,E1 20937.88,E2 20937.88} C_VEL
LIN {X 0,Y 452.235,Z 1054.375,A -85,B 0,C 180,E1 20937.071,E2 20937.071} C_VEL
LIN {X 0,Y 453.219,Z 1033.154,A -85,B 0,C 180,E1 20936.49,E2 20936.49} C_VEL
LIN {X 0,Y 458.642,Z 802.182,A -85,B 0,C 180,E1 20932.538,E2 20932.538} C_VEL
LIN {X 0,Y 452.435,Z 774.456,A -85,B 0,C 180,E1 20931.362,E2 20931.362} C_VEL
LIN {X 0,Y 453.869,Z 746.576,A -85,B 0,C 180,E1 20928.463,E2 20928.463} C_VEL
LIN {X 0,Y 454.618,Z 734.171,A -85,B 0,C 180,E1 20927.087,E2 20927.087} C_VEL
LIN {X 0,Y 448.245,Z 715.868,A -85,B 0,C 180,E1 20924.089,E2 20924.089} C_VEL
LIN {X 0,Y 443.41,Z 703.64,A -85,B 0,C 180,E1 20921.915,E2 20921.915} C_VEL
LIN {X 0,Y 450.767,Z 721.528,A -85,B 0,C 180,E1 20918.972,E2 20918.972} C_VEL
LIN {X 0,Y 455.095,Z 733.456,A -85,B 0,C 180,E1 20917.17,E2 20917.17} C_VEL
LIN {X 0,Y 451.672,Z 771.519,A -85,B 0,C 180,E1 20913.43,E2 20913.43} C_VEL
LIN {X 0,Y 448.266,Z 812.646,A -85,B 0,C 180,E1 20909.461,E2 20909.461} C_VEL
LIN {X 0,Y 445.195,Z 853.83,A -85,B 0,C 180,E1 20905.545,E2 20905.545} C_VEL
LIN {X 0,Y 445.044,Z 857.966,A -85,B 0,C 180,E1 20905.188,E2 20905.188} C_VEL
LIN {X 0,Y 446.268,Z 867.471,A -85,B 0,C 180,E1 20904.889,E2 20904.889} C_VEL
LIN {X 0,Y 441.883,Z 1028.766,A -85,B 0,C 180,E1 20901.674,E2 20901.674} C_VEL
LIN {X 0,Y 441.31,Z 1046.792,A -85,B 0,C 180,E1 20901.053,E2 20901.053} C_VEL
LIN {X 0,Y 440.527,Z 1063.206,A -85,B 0,C 180,E1 20900.251,E2 20900.251} C_VEL
LIN {X 0,Y 439.515,Z 1079.532,A -85,B 0,C 180,E1 20899.192,E2 20899.192} C_VEL
LIN {X 0,Y 438.388,Z 1094.692,A -85,B 0,C 180,E1 20897.933,E2 20897.933} C_VEL
LIN {X 0,Y 437.249,Z 1108.859,A -85,B 0,C 180,E1 20896.473,E2 20896.473} C_VEL
LIN {X 0,Y 436.171,Z 1121.475,A -85,B 0,C 180,E1 20894.877,E2 20894.877} C_VEL
LIN {X 0,Y 435.143,Z 1133.289,A -85,B 0,C 180,E1 20893.028,E2 20893.028} C_VEL
LIN {X 0,Y 434.268,Z 1143.684,A -85,B 0,C 180,E1 20891.017,E2 20891.017} C_VEL
LIN {X 0,Y 433.618,Z 1152.423,A -85,B 0,C 180,E1 20888.888,E2 20888.888} C_VEL
LIN {X 0,Y 433.204,Z 1159.113,A -85,B 0,C 180,E1 20886.76,E2 20886.76} C_VEL
LIN {X 0,Y 432.927,Z 1164.369,A -85,B 0,C 180,E1 20884.504,E2 20884.504} C_VEL
LIN {X 0,Y 432.821,Z 1167.883,A -85,B 0,C 180,E1 20882.251,E2 20882.251} C_VEL
LIN {X 0,Y 432.794,Z 1169.749,A -85,B 0,C 180,E1 20880,E2 20880} C_VEL
LIN {X 0,Y 432.844,Z 1169.958,A -85,B 0,C 180,E1 20877.75,E2 20877.75} C_VEL
LIN {X 0,Y 432.988,Z 1168.461,A -85,B 0,C 180,E1 20875.364,E2 20875.364} C_VEL
LIN {X 0,Y 433.25,Z 1165.386,A -85,B 0,C 180,E1 20873.108,E2 20873.108} C_VEL
LIN {X 0,Y 433.666,Z 1160.501,A -85,B 0,C 180,E1 20870.846,E2 20870.846} C_VEL
LIN {X 0,Y 434.283,Z 1153.689,A -85,B 0,C 180,E1 20868.58,E2 20868.58} C_VEL
LIN {X 0,Y 435.097,Z 1145.836,A -85,B 0,C 180,E1 20866.58,E2 20866.58} C_VEL
LIN {X 0,Y 436.146,Z 1135.818,A -85,B 0,C 180,E1 20864.578,E2 20864.578} C_VEL
LIN {X 0,Y 437.235,Z 1125.059,A -85,B 0,C 180,E1 20862.843,E2 20862.843} C_VEL
LIN {X 0,Y 438.428,Z 1112.867,A -85,B 0,C 180,E1 20861.243,E2 20861.243} C_VEL
LIN {X 0,Y 439.6,Z 1099.359,A -85,B 0,C 180,E1 20859.822,E2 20859.822} C_VEL
LIN {X 0,Y 440.702,Z 1084.545,A -85,B 0,C 180,E1 20858.576,E2 20858.576} C_VEL
LIN {X 0,Y 441.573,Z 1069.292,A -85,B 0,C 180,E1 20857.571,E2 20857.571} C_VEL
LIN {X 0,Y 442.208,Z 1052.587,A -85,B 0,C 180,E1 20856.762,E2 20856.762} C_VEL
LIN {X 0,Y 442.551,Z 1035.572,A -85,B 0,C 180,E1 20856.193,E2 20856.193} C_VEL
LIN {X 0,Y 444.226,Z 991.046,A -85,B 0,C 180,E1 20855.078,E2 20855.078} C_VEL
LIN {X 0,Y 449.328,Z 913.932,A -85,B 0,C 180,E1 20852.999,E2 20852.999} C_VEL
LIN {X 0,Y 451.494,Z 888.812,A -85,B 0,C 180,E1 20852.286,E2 20852.286} C_VEL
LIN {X 0,Y 458.142,Z 873.623,A -85,B 0,C 180,E1 20851.164,E2 20851.164} C_VEL
LIN {X 0,Y 464.684,Z 850.644,A -85,B 0,C 180,E1 20848.331,E2 20848.331} C_VEL
LIN {X 0,Y 471.837,Z 832.787,A -85,B 0,C 180,E1 20845.951,E2 20845.951} C_VEL
LIN {X 0,Y 478.238,Z 820.966,A -85,B 0,C 180,E1 20844.213,E2 20844.213} C_VEL
LIN {X 0,Y 472.836,Z 829.781,A -85,B 0,C 180,E1 20842.788,E2 20842.788} C_VEL
LIN {X 0,Y 469.737,Z 838.419,A -85,B 0,C 180,E1 20841.369,E2 20841.369} C_VEL
LIN {X 0,Y 468.771,Z 847.491,A -85,B 0,C 180,E1 20839.899,E2 20839.899} C_VEL
LIN {X 0,Y 470.033,Z 856.937,A -85,B 0,C 180,E1 20838.419,E2 20838.419} C_VEL
LIN {X 0,Y 473.694,Z 866.913,A -85,B 0,C 180,E1 20836.914,E2 20836.914} C_VEL
LIN {X 0,Y 479.523,Z 876.698,A -85,B 0,C 180,E1 20835.489,E2 20835.489} C_VEL
LIN {X 0,Y 487.509,Z 886.345,A -85,B 0,C 180,E1 20834.125,E2 20834.125} C_VEL
LIN {X 0,Y 497.704,Z 895.623,A -85,B 0,C 180,E1 20832.84,E2 20832.84} C_VEL
LIN {X 0,Y 507.262,Z 902.799,A -85,B 0,C 180,E1 20831.874,E2 20831.874} C_VEL
LIN {X 0,Y 491.908,Z 926.868,A -85,B 0,C 180,E1 20831.269,E2 20831.269} C_VEL
LIN {X 0,Y 481.611,Z 945.757,A -85,B 0,C 180,E1 20830.684,E2 20830.684} C_VEL
LIN {X 0,Y 474.516,Z 961.998,A -85,B 0,C 180,E1 20830.07,E2 20830.07} C_VEL
LIN {X 0,Y 465.723,Z 980.745,A -85,B 0,C 180,E1 20829.376,E2 20829.376} C_VEL
LIN {X 0,Y 456.522,Z 1006.811,A -85,B 0,C 180,E1 20828.243,E2 20828.243} C_VEL
LIN {X 0,Y 454.199,Z 1026.337,A -85,B 0,C 180,E1 20828.023,E2 20828.023} C_VEL
LIN {X 0,Y 453.271,Z 1055.998,A -85,B 0,C 180,E1 20827.429,E2 20827.429} C_VEL
LIN {X 0,Y 451.726,Z 1081.468,A -85,B 0,C 180,E1 20826.687,E2 20826.687} C_VEL
LIN {X 0,Y 450.05,Z 1105.945,A -85,B 0,C 180,E1 20825.728,E2 20825.728} C_VEL
LIN {X 0,Y 448.258,Z 1128.926,A -85,B 0,C 180,E1 20824.589,E2 20824.589} C_VEL
LIN {X 0,Y 446.301,Z 1151.427,A -85,B 0,C 180,E1 20823.214,E2 20823.214} C_VEL
LIN {X 0,Y 444.328,Z 1173.072,A -85,B 0,C 180,E1 20821.622,E2 20821.622} C_VEL
LIN {X 0,Y 442.356,Z 1192.913,A -85,B 0,C 180,E1 20819.894,E2 20819.894} C_VEL
LIN {X 0,Y 440.422,Z 1211.523,A -85,B 0,C 180,E1 20817.98,E2 20817.98} C_VEL
LIN {X 0,Y 438.718,Z 1227.609,A -85,B 0,C 180,E1 20816.033,E2 20816.033} C_VEL
LIN {X 0,Y 437.217,Z 1241.663,A -85,B 0,C 180,E1 20814.068,E2 20814.068} C_VEL
LIN {X 0,Y 435.764,Z 1255.569,A -85,B 0,C 180,E1 20811.821,E2 20811.821} C_VEL
LIN {X 0,Y 434.56,Z 1267.683,A -85,B 0,C 180,E1 20809.489,E2 20809.489} C_VEL
LIN {X 0,Y 433.689,Z 1277.171,A -85,B 0,C 180,E1 20807.358,E2 20807.358} C_VEL
LIN {X 0,Y 433.034,Z 1285.169,A -85,B 0,C 180,E1 20805.262,E2 20805.262} C_VEL
LIN {X 0,Y 432.526,Z 1292.561,A -85,B 0,C 180,E1 20802.958,E2 20802.958} C_VEL
LIN {X 0,Y 432.177,Z 1299.119,A -85,B 0,C 180,E1 20800.262,E2 20800.262} C_VEL
LIN {X 0,Y 431.991,Z 1303.779,A -85,B 0,C 180,E1 20797.582,E2 20797.582} C_VEL
LIN {X 0,Y 431.923,Z 1306.783,A -85,B 0,C 180,E1 20795.18,E2 20795.18} C_VEL
LIN {X 0,Y 431.902,Z 1308.659,A -85,B 0,C 180,E1 20792.787,E2 20792.787} C_VEL
LIN {X 0,Y 431.907,Z 1309.484,A -85,B 0,C 180,E1 20789.868,E2 20789.868} C_VEL
LIN {X 0,Y 431.903,Z 1308.578,A -85,B 0,C 180,E1 20787.081,E2 20787.081} C_VEL
LIN {X 0,Y 431.927,Z 1306.645,A -85,B 0,C 180,E1 20784.688,E2 20784.688} C_VEL
LIN {X 0,Y 432.002,Z 1303.581,A -85,B 0,C 180,E1 20782.286,E2 20782.286} C_VEL
LIN {X 0,Y 432.202,Z 1298.594,A -85,B 0,C 180,E1 20779.47,E2 20779.47} C_VEL
LIN {X 0,Y 432.547,Z 1292.172,A -85,B 0,C 180,E1 20776.908,E2 20776.908} C_VEL
LIN {X 0,Y 433.067,Z 1284.864,A -85,B 0,C 180,E1 20774.603,E2 20774.603} C_VEL
LIN {X 0,Y 433.752,Z 1276.721,A -85,B 0,C 180,E1 20772.425,E2 20772.425} C_VEL
LIN {X 0,Y 434.816,Z 1265.986,A -85,B 0,C 180,E1 20769.964,E2 20769.964} C_VEL
LIN {X 0,Y 436.267,Z 1252.423,A -85,B 0,C 180,E1 20767.355,E2 20767.355} C_VEL
LIN {X 0,Y 437.851,Z 1239.07,A -85,B 0,C 180,E1 20765.155,E2 20765.155} C_VEL
LIN {X 0,Y 439.9,Z 1222.629,A -85,B 0,C 180,E1 20762.816,E2 20762.816} C_VEL
LIN {X 0,Y 442.129,Z 1204.946,A -85,B 0,C 180,E1 20760.686,E2 20760.686} C_VEL
LIN {X 0,Y 444.534,Z 1185.962,A -85,B 0,C 180,E1 20758.727,E2 20758.727} C_VEL
LIN {X 0,Y 446.942,Z 1166.419,A -85,B 0,C 180,E1 20757.025,E2 20757.025} C_VEL
LIN {X 0,Y 449.479,Z 1144.791,A -85,B 0,C 180,E1 20755.443,E2 20755.443} C_VEL
LIN {X 0,Y 451.919,Z 1122.451,A -85,B 0,C 180,E1 20754.106,E2 20754.106} C_VEL
LIN {X 0,Y 454.05,Z 1100.141,A -85,B 0,C 180,E1 20753.047,E2 20753.047} C_VEL
LIN {X 0,Y 455.995,Z 1076.494,A -85,B 0,C 180,E1 20752.194,E2 20752.194} C_VEL
LIN {X 0,Y 457.44,Z 1052.808,A -85,B 0,C 180,E1 20751.594,E2 20751.594} C_VEL
LIN {X 0,Y 458.722,Z 1021.326,A -85,B 0,C 180,E1 20751.024,E2 20751.024} C_VEL
LIN {X 0,Y 459.345,Z 1016.323,A -85,B 0,C 180,E1 20750.939,E2 20750.939} C_VEL
LIN {X 0,Y 464.755,Z 1000.736,A -85,B 0,C 180,E1 20750.207,E2 20750.207} C_VEL
LIN {X 0,Y 470.987,Z 984.299,A -85,B 0,C 180,E1 20749.489,E2 20749.489} C_VEL
LIN {X 0,Y 479.866,Z 965.44,A -85,B 0,C 180,E1 20748.821,E2 20748.821} C_VEL
LIN {X 0,Y 487.164,Z 949.274,A -85,B 0,C 180,E1 20748.241,E2 20748.241} C_VEL
LIN {X 0,Y 497.895,Z 929.252,A -85,B 0,C 180,E1 20747.722,E2 20747.722} C_VEL
LIN {X 0,Y 511.48,Z 906.728,A -85,B 0,C 180,E1 20747.288,E2 20747.288} C_VEL
LIN {X 0,Y 500.258,Z 898.345,A -85,B 0,C 180,E1 20745.686,E2 20745.686} C_VEL
LIN {X 0,Y 491.28,Z 888.972,A -85,B 0,C 180,E1 20744.11,E2 20744.11} C_VEL
LIN {X 0,Y 483.853,Z 878.211,A -85,B 0,C 180,E1 20742.51,E2 20742.51} C_VEL
LIN {X 0,Y 477.825,Z 865.524,A -85,B 0,C 180,E1 20740.837,E2 20740.837} C_VEL
LIN {X 0,Y 473.683,Z 851.891,A -85,B 0,C 180,E1 20739.226,E2 20739.226} C_VEL
LIN {X 0,Y 471.164,Z 836.588,A -85,B 0,C 180,E1 20737.597,E2 20737.597} C_VEL
LIN {X 0,Y 470.35,Z 818.968,A -85,B 0,C 180,E1 20735.913,E2 20735.913} C_VEL
LIN {X 0,Y 471.573,Z 797.643,A -85,B 0,C 180,E1 20734.111,E2 20734.111} C_VEL
LIN {X 0,Y 476.09,Z 758.476,A -85,B 0,C 180,E1 20730.985,E2 20730.985} C_VEL
LIN {X 0,Y 465.94,Z 739.08,A -85,B 0,C 180,E1 20727.475,E2 20727.475} C_VEL
LIN {X 0,Y 457.165,Z 723.237,A -85,B 0,C 180,E1 20724.278,E2 20724.278} C_VEL
LIN {X 0,Y 450.019,Z 710.478,A -85,B 0,C 180,E1 20721.506,E2 20721.506} C_VEL
LIN {X 0,Y 444.297,Z 700.544,A -85,B 0,C 180,E1 20719.181,E2 20719.181} C_VEL
LIN {X 0,Y 441.381,Z 695.517,A -85,B 0,C 180,E1 20717.943,E2 20717.943} C_VEL
LIN {X 0,Y 438.531,Z 690.567,A -85,B 0,C 180,E1 20716.695,E2 20716.695} C_VEL
LIN {X 0,Y 436.544,Z 687.2,A -85,B 0,C 180,E1 20715.816,E2 20715.816} C_VEL
LIN {X 0,Y 435.765,Z 685.644,A -85,B 0,C 180,E1 20715.436,E2 20715.436} C_VEL
LIN {X 0,Y 433.707,Z 682.582,A -85,B 0,C 180,E1 20714.553,E2 20714.553} C_VEL
LIN {X 0,Y 433.248,Z 680.766,A -85,B 0,C 180,E1 20714.16,E2 20714.16} C_VEL
LIN {X 0,Y 433.258,Z 680.764,A -85,B 0,C 180,E1 20710.37,E2 20710.37} C_VEL
LIN {X 0,Y 433.245,Z 680.764,A -85,B 0,C 180,E1 20706.493,E2 20706.493} C_VEL
LIN {X 0,Y 433.25,Z 680.765,A -85,B 0,C 180,E1 20702.778,E2 20702.778} C_VEL
LIN {X 0,Y 433.248,Z 680.768,A -85,B 0,C 180,E1 20699.074,E2 20699.074} C_VEL
LIN {X 0,Y 433.255,Z 680.767,A -85,B 0,C 180,E1 20695.234,E2 20695.234} C_VEL
LIN {X 0,Y 433.248,Z 680.765,A -85,B 0,C 180,E1 20691.506,E2 20691.506} C_VEL
LIN {X 0,Y 433.255,Z 680.768,A -85,B 0,C 180,E1 20687.742,E2 20687.742} C_VEL
LIN {X 0,Y 433.257,Z 680.765,A -85,B 0,C 180,E1 20683.922,E2 20683.922} C_VEL
LIN {X 0,Y 433.255,Z 680.759,A -85,B 0,C 180,E1 20680.028,E2 20680.028} C_VEL
LIN {X 0,Y 433.254,Z 680.757,A -85,B 0,C 180,E1 20676.324,E2 20676.324} C_VEL
LIN {X 0,Y 433.256,Z 680.73,A -85,B 0,C 180,E1 20672.512,E2 20672.512} C_VEL
LIN {X 0,Y 433.265,Z 680.76,A -85,B 0,C 180,E1 20668.564,E2 20668.564} C_VEL
LIN {X 0,Y 433.245,Z 680.724,A -85,B 0,C 180,E1 20664.763,E2 20664.763} C_VEL
LIN {X 0,Y 433.257,Z 680.755,A -85,B 0,C 180,E1 20660.948,E2 20660.948} C_VEL
LIN {X 0,Y 433.258,Z 680.806,A -85,B 0,C 180,E1 20658.722,E2 20658.722} C_VEL
LIN {X 0,Y 434.357,Z 683.905,A -85,B 0,C 180,E1 20658.298,E2 20658.298} C_VEL
LIN {X 0,Y 435.894,Z 686.424,A -85,B 0,C 180,E1 20657.86,E2 20657.86} C_VEL
LIN {X 0,Y 443.988,Z 702.487,A -85,B 0,C 180,E1 20655.362,E2 20655.362} C_VEL
LIN {X 0,Y 452.245,Z 720.868,A -85,B 0,C 180,E1 20652.776,E2 20652.776} C_VEL
LIN {X 0,Y 457.63,Z 734.59,A -85,B 0,C 180,E1 20651.009,E2 20651.009} C_VEL
LIN {X 0,Y 455.767,Z 770.563,A -85,B 0,C 180,E1 20648.377,E2 20648.377} C_VEL
LIN {X 0,Y 455.892,Z 773.807,A -85,B 0,C 180,E1 20648.196,E2 20648.196} C_VEL
LIN {X 0,Y 458.809,Z 794.778,A -85,B 0,C 180,E1 20647.496,E2 20647.496} C_VEL
LIN {X 0,Y 455.183,Z 947.878,A -85,B 0,C 180,E1 20644.89,E2 20644.89} C_VEL
LIN {X 0,Y 454.216,Z 955.566,A -85,B 0,C 180,E1 20644.83,E2 20644.83} C_VEL
LIN {X 0,Y 448.639,Z 976.052,A -85,B 0,C 180,E1 20644.939,E2 20644.939} C_VEL
LIN {X 0,Y 447.843,Z 982.654,A -85,B 0,C 180,E1 20644.884,E2 20644.884} C_VEL
LIN {X 0,Y 446.488,Z 1036.151,A -85,B 0,C 180,E1 20643.928,E2 20643.928} C_VEL
LIN {X 0,Y 445.448,Z 1056.476,A -85,B 0,C 180,E1 20643.342,E2 20643.342} C_VEL
LIN {X 0,Y 444.014,Z 1076.588,A -85,B 0,C 180,E1 20642.522,E2 20642.522} C_VEL
LIN {X 0,Y 442.21,Z 1095.985,A -85,B 0,C 180,E1 20641.486,E2 20641.486} C_VEL
LIN {X 0,Y 440.235,Z 1114.043,A -85,B 0,C 180,E1 20640.278,E2 20640.278} C_VEL
LIN {X 0,Y 437.983,Z 1132.126,A -85,B 0,C 180,E1 20638.795,E2 20638.795} C_VEL
LIN {X 0,Y 435.55,Z 1149.752,A -85,B 0,C 180,E1 20637.034,E2 20637.034} C_VEL
LIN {X 0,Y 433.213,Z 1165.575,A -85,B 0,C 180,E1 20635.129,E2 20635.129} C_VEL
LIN {X 0,Y 431.079,Z 1179.875,A -85,B 0,C 180,E1 20633.077,E2 20633.077} C_VEL
LIN {X 0,Y 429.177,Z 1192.776,A -85,B 0,C 180,E1 20630.881,E2 20630.881} C_VEL
LIN {X 0,Y 427.476,Z 1204.931,A -85,B 0,C 180,E1 20628.406,E2 20628.406} C_VEL
LIN {X 0,Y 426.174,Z 1215.237,A -85,B 0,C 180,E1 20625.863,E2 20625.863} C_VEL
LIN {X 0,Y 425.229,Z 1223.925,A -85,B 0,C 180,E1 20623.23,E2 20623.23} C_VEL
LIN {X 0,Y 424.623,Z 1230.868,A -85,B 0,C 180,E1 20620.583,E2 20620.583} C_VEL
LIN {X 0,Y 424.271,Z 1236.225,A -85,B 0,C 180,E1 20617.855,E2 20617.855} C_VEL
LIN {X 0,Y 424.097,Z 1239.929,A -85,B 0,C 180,E1 20615.139,E2 20615.139} C_VEL
LIN {X 0,Y 424.041,Z 1242.149,A -85,B 0,C 180,E1 20612.297,E2 20612.297} C_VEL
LIN {X 0,Y 424.026,Z 1242.723,A -85,B 0,C 180,E1 20609.594,E2 20609.594} C_VEL
LIN {X 0,Y 424.052,Z 1241.803,A -85,B 0,C 180,E1 20606.891,E2 20606.891} C_VEL
LIN {X 0,Y 424.126,Z 1239.273,A -85,B 0,C 180,E1 20604.181,E2 20604.181} C_VEL
LIN {X 0,Y 424.319,Z 1235.171,A -85,B 0,C 180,E1 20601.462,E2 20601.462} C_VEL
LIN {X 0,Y 424.725,Z 1229.402,A -85,B 0,C 180,E1 20598.732,E2 20598.732} C_VEL
LIN {X 0,Y 425.396,Z 1222.179,A -85,B 0,C 180,E1 20596.102,E2 20596.102} C_VEL
LIN {X 0,Y 426.413,Z 1213.307,A -85,B 0,C 180,E1 20593.517,E2 20593.517} C_VEL
LIN {X 0,Y 427.857,Z 1202.255,A -85,B 0,C 180,E1 20590.903,E2 20590.903} C_VEL
LIN {X 0,Y 429.664,Z 1189.53,A -85,B 0,C 180,E1 20588.427,E2 20588.427} C_VEL
LIN {X 0,Y 431.724,Z 1175.62,A -85,B 0,C 180,E1 20586.179,E2 20586.179} C_VEL
LIN {X 0,Y 433.917,Z 1160.874,A -85,B 0,C 180,E1 20584.182,E2 20584.182} C_VEL
LIN {X 0,Y 436.235,Z 1144.733,A -85,B 0,C 180,E1 20582.345,E2 20582.345} C_VEL
LIN {X 0,Y 438.545,Z 1127.614,A -85,B 0,C 180,E1 20580.722,E2 20580.722} C_VEL
LIN {X 0,Y 440.755,Z 1109.561,A -85,B 0,C 180,E1 20579.308,E2 20579.308} C_VEL
LIN {X 0,Y 442.767,Z 1090.735,A -85,B 0,C 180,E1 20578.113,E2 20578.113} C_VEL
LIN {X 0,Y 444.474,Z 1071.145,A -85,B 0,C 180,E1 20577.132,E2 20577.132} C_VEL
LIN {X 0,Y 445.842,Z 1050.521,A -85,B 0,C 180,E1 20576.367,E2 20576.367} C_VEL
LIN {X 0,Y 446.691,Z 1030.255,A -85,B 0,C 180,E1 20575.853,E2 20575.853} C_VEL
LIN {X 0,Y 452.295,Z 803.751,A -85,B 0,C 180,E1 20571.942,E2 20571.942} C_VEL
LIN {X 0,Y 445.911,Z 774.877,A -85,B 0,C 180,E1 20570.678,E2 20570.678} C_VEL
LIN {X 0,Y 447.434,Z 746.766,A -85,B 0,C 180,E1 20567.729,E2 20567.729} C_VEL
LIN {X 0,Y 447.91,Z 737.636,A -85,B 0,C 180,E1 20566.696,E2 20566.696} C_VEL
LIN {X 0,Y 441.321,Z 718.658,A -85,B 0,C 180,E1 20563.531,E2 20563.531} C_VEL
LIN {X 0,Y 437.789,Z 709.718,A -85,B 0,C 180,E1 20561.916,E2 20561.916} C_VEL
LIN {X 0,Y 445.171,Z 727.964,A -85,B 0,C 180,E1 20558.9,E2 20558.9} C_VEL
LIN {X 0,Y 448.352,Z 736.674,A -85,B 0,C 180,E1 20557.562,E2 20557.562} C_VEL
LIN {X 0,Y 444.802,Z 774.617,A -85,B 0,C 180,E1 20553.804,E2 20553.804} C_VEL
LIN {X 0,Y 441.241,Z 815.461,A -85,B 0,C 180,E1 20549.82,E2 20549.82} C_VEL
LIN {X 0,Y 438.095,Z 855.878,A -85,B 0,C 180,E1 20545.944,E2 20545.944} C_VEL
LIN {X 0,Y 438.016,Z 859.152,A -85,B 0,C 180,E1 20545.673,E2 20545.673} C_VEL
LIN {X 0,Y 439.226,Z 868.655,A -85,B 0,C 180,E1 20545.368,E2 20545.368} C_VEL
LIN {X 0,Y 434.496,Z 1029.719,A -85,B 0,C 180,E1 20542.062,E2 20542.062} C_VEL
LIN {X 0,Y 433.904,Z 1047.586,A -85,B 0,C 180,E1 20541.436,E2 20541.436} C_VEL
LIN {X 0,Y 433.08,Z 1064.136,A -85,B 0,C 180,E1 20540.615,E2 20540.615} C_VEL
LIN {X 0,Y 432.091,Z 1079.626,A -85,B 0,C 180,E1 20539.605,E2 20539.605} C_VEL
LIN {X 0,Y 430.905,Z 1094.984,A -85,B 0,C 180,E1 20538.325,E2 20538.325} C_VEL
LIN {X 0,Y 429.646,Z 1109.903,A -85,B 0,C 180,E1 20536.773,E2 20536.773} C_VEL
LIN {X 0,Y 428.512,Z 1122.567,A -85,B 0,C 180,E1 20535.149,E2 20535.149} C_VEL
LIN {X 0,Y 427.457,Z 1134.091,A -85,B 0,C 180,E1 20533.329,E2 20533.329} C_VEL
LIN {X 0,Y 426.497,Z 1144.867,A -85,B 0,C 180,E1 20531.221,E2 20531.221} C_VEL
LIN {X 0,Y 425.801,Z 1153.651,A -85,B 0,C 180,E1 20529.052,E2 20529.052} C_VEL
LIN {X 0,Y 425.333,Z 1160.74,A -85,B 0,C 180,E1 20526.75,E2 20526.75} C_VEL
LIN {X 0,Y 425.049,Z 1165.94,A -85,B 0,C 180,E1 20524.452,E2 20524.452} C_VEL
LIN {X 0,Y 424.941,Z 1169.4,A -85,B 0,C 180,E1 20522.158,E2 20522.158} C_VEL
LIN {X 0,Y 424.909,Z 1171.171,A -85,B 0,C 180,E1 20519.865,E2 20519.865} C_VEL
LIN {X 0,Y 424.992,Z 1171.289,A -85,B 0,C 180,E1 20517.438,E2 20517.438} C_VEL
LIN {X 0,Y 425.165,Z 1169.67,A -85,B 0,C 180,E1 20515.009,E2 20515.009} C_VEL
LIN {X 0,Y 425.486,Z 1166.372,A -85,B 0,C 180,E1 20512.71,E2 20512.71} C_VEL
LIN {X 0,Y 425.971,Z 1161.163,A -85,B 0,C 180,E1 20510.349,E2 20510.349} C_VEL
LIN {X 0,Y 426.693,Z 1154.33,A -85,B 0,C 180,E1 20508.1,E2 20508.1} C_VEL
LIN {X 0,Y 427.625,Z 1145.96,A -85,B 0,C 180,E1 20506.011,E2 20506.011} C_VEL
LIN {X 0,Y 428.764,Z 1135.959,A -85,B 0,C 180,E1 20504.028,E2 20504.028} C_VEL
LIN {X 0,Y 429.973,Z 1124.915,A -85,B 0,C 180,E1 20502.265,E2 20502.265} C_VEL
LIN {X 0,Y 431.266,Z 1112.261,A -85,B 0,C 180,E1 20500.638,E2 20500.638} C_VEL
LIN {X 0,Y 432.519,Z 1098.565,A -85,B 0,C 180,E1 20499.216,E2 20499.216} C_VEL
LIN {X 0,Y 433.648,Z 1083.659,A -85,B 0,C 180,E1 20497.989,E2 20497.989} C_VEL
LIN {X 0,Y 434.553,Z 1067.695,A -85,B 0,C 180,E1 20496.974,E2 20496.974} C_VEL
LIN {X 0,Y 435.176,Z 1051.435,A -85,B 0,C 180,E1 20496.211,E2 20496.211} C_VEL
LIN {X 0,Y 435.541,Z 1031.409,A -85,B 0,C 180,E1 20495.588,E2 20495.588} C_VEL
LIN {X 0,Y 438.263,Z 979.424,A -85,B 0,C 180,E1 20494.184,E2 20494.184} C_VEL
LIN {X 0,Y 445.309,Z 893.323,A -85,B 0,C 180,E1 20491.703,E2 20491.703} C_VEL
LIN {X 0,Y 453.068,Z 876.285,A -85,B 0,C 180,E1 20490.447,E2 20490.447} C_VEL
LIN {X 0,Y 460.052,Z 854.513,A -85,B 0,C 180,E1 20487.68,E2 20487.68} C_VEL
LIN {X 0,Y 467.295,Z 838.312,A -85,B 0,C 180,E1 20485.458,E2 20485.458} C_VEL
LIN {X 0,Y 472.114,Z 829.97,A -85,B 0,C 180,E1 20484.207,E2 20484.207} C_VEL
LIN {X 0,Y 466.971,Z 838.743,A -85,B 0,C 180,E1 20482.703,E2 20482.703} C_VEL
LIN {X 0,Y 464.237,Z 847.271,A -85,B 0,C 180,E1 20481.23,E2 20481.23} C_VEL
LIN {X 0,Y 463.693,Z 856.325,A -85,B 0,C 180,E1 20479.693,E2 20479.693} C_VEL
LIN {X 0,Y 465.386,Z 865.453,A -85,B 0,C 180,E1 20478.204,E2 20478.204} C_VEL
LIN {X 0,Y 469.398,Z 875.074,A -85,B 0,C 180,E1 20476.695,E2 20476.695} C_VEL
LIN {X 0,Y 475.661,Z 884.723,A -85,B 0,C 180,E1 20475.237,E2 20475.237} C_VEL
LIN {X 0,Y 483.967,Z 894.15,A -85,B 0,C 180,E1 20473.862,E2 20473.862} C_VEL
